LIN {X 0,Y 421.841,Z 771.476,A -85,B 0,C 180,E1 10209.107,E2 10209.107} C_VEL
LIN {X 0,Y 405.011,Z 742.574,A -85,B 0,C 180,E1 10212.582,E2 10212.582} C_VEL
LIN {X 0,Y 403.08,Z 737.44,A -85,B 0,C 180,E1 10213.086,E2 10213.086} C_VEL
LIN {X 0,Y 403.121,Z 737.44,A -85,B 0,C 180,E1 10218.689,E2 10218.689} C_VEL
LIN {X 0,Y 403.149,Z 737.44,A -85,B 0,C 180,E1 10225.725,E2 10225.725} C_VEL
LIN {X 0,Y 403.287,Z 737.44,A -85,B 0,C 180,E1 10230.797,E2 10230.797} C_VEL
LIN {X 0,Y 403.605,Z 737.44,A -85,B 0,C 180,E1 10237.976,E2 10237.976} C_VEL
LIN {X 0,Y 403.898,Z 737.44,A -85,B 0,C 180,E1 10244.795,E2 10244.795} C_VEL
LIN {X 0,Y 404.153,Z 737.44,A -85,B 0,C 180,E1 10251.389,E2 10251.389} C_VEL
LIN {X 0,Y 404.396,Z 737.44,A -85,B 0,C 180,E1 10257.86,E2 10257.86} C_VEL
LIN {X 0,Y 404.246,Z 737.44,A -85,B 0,C 180,E1 10264.301,E2 10264.301} C_VEL
LIN {X 0,Y 403.948,Z 737.44,A -85,B 0,C 180,E1 10270.806,E2 10270.806} C_VEL
LIN {X 0,Y 403.703,Z 737.44,A -85,B 0,C 180,E1 10277.463,E2 10277.463} C_VEL
LIN {X 0,Y 403.474,Z 737.44,A -85,B 0,C 180,E1 10284.383,E2 10284.383} C_VEL
LIN {X 0,Y 403.248,Z 737.44,A -85,B 0,C 180,E1 10291.714,E2 10291.714} C_VEL
LIN {X 0,Y 403.323,Z 738.232,A -85,B 0,C 180,E1 10296.977,E2 10296.977} C_VEL
LIN {X 0,Y 406.403,Z 743.737,A -85,B 0,C 180,E1 10297.606,E2 10297.606} C_VEL
LIN {X 0,Y 427.744,Z 781.818,A -85,B 0,C 180,E1 10301.54,E2 10301.54} C_VEL
LIN {X 0,Y 442.603,Z 815.8,A -85,B 0,C 180,E1 10304.217,E2 10304.217} C_VEL
LIN {X 0,Y 438.64,Z 858.115,A -85,B 0,C 180,E1 10305.69,E2 10305.69} C_VEL
LIN {X 0,Y 433.492,Z 898.592,A -85,B 0,C 180,E1 10307.86,E2 10307.86} C_VEL
LIN {X 0,Y 427.452,Z 938.526,A -85,B 0,C 180,E1 10310.854,E2 10310.854} C_VEL
LIN {X 0,Y 420.959,Z 978.52,A -85,B 0,C 180,E1 10314.869,E2 10314.869} C_VEL
LIN {X 0,Y 415.665,Z 1011.15,A -85,B 0,C 180,E1 10319.101,E2 10319.101} C_VEL
LIN {X 0,Y 411.27,Z 1038.766,A -85,B 0,C 180,E1 10323.784,E2 10323.784} C_VEL
LIN {X 0,Y 408.924,Z 1055.24,A -85,B 0,C 180,E1 10327.316,E2 10327.316} C_VEL
LIN {X 0,Y 403.983,Z 1063.313,A -85,B 0,C 180,E1 10329.395,E2 10329.395} C_VEL
LIN {X 0,Y 399.077,Z 1070.528,A -85,B 0,C 180,E1 10331.574,E2 10331.574} C_VEL
LIN {X 0,Y 397.48,Z 1085.683,A -85,B 0,C 180,E1 10337.349,E2 10337.349} C_VEL
LIN {X 0,Y 396.899,Z 1094.4,A -85,B 0,C 180,E1 10342.658,E2 10342.658} C_VEL
LIN {X 0,Y 396.783,Z 1098.451,A -85,B 0,C 180,E1 10347.813,E2 10347.813} C_VEL
LIN {X 0,Y 396.696,Z 1098.441,A -85,B 0,C 180,E1 10352.187,E2 10352.187} C_VEL
LIN {X 0,Y 396.89,Z 1094.411,A -85,B 0,C 180,E1 10357.332,E2 10357.332} C_VEL
LIN {X 0,Y 397.455,Z 1085.675,A -85,B 0,C 180,E1 10362.652,E2 10362.652} C_VEL
LIN {X 0,Y 398.842,Z 1071.644,A -85,B 0,C 180,E1 10368.064,E2 10368.064} C_VEL
LIN {X 0,Y 401.384,Z 1052.51,A -85,B 0,C 180,E1 10373.331,E2 10373.331} C_VEL
LIN {X 0,Y 405.144,Z 1028.089,A -85,B 0,C 180,E1 10378.34,E2 10378.34} C_VEL
LIN {X 0,Y 410.502,Z 996.087,A -85,B 0,C 180,E1 10383.284,E2 10383.284} C_VEL
LIN {X 0,Y 417.164,Z 957.356,A -85,B 0,C 180,E1 10387.871,E2 10387.871} C_VEL
LIN {X 0,Y 423.856,Z 917.641,A -85,B 0,C 180,E1 10391.397,E2 10391.397} C_VEL
LIN {X 0,Y 430,Z 877.022,A -85,B 0,C 180,E1 10394.013,E2 10394.013} C_VEL
LIN {X 0,Y 435.089,Z 835.418,A -85,B 0,C 180,E1 10395.826,E2 10395.826} C_VEL
LIN {X 0,Y 436.104,Z 818.323,A -85,B 0,C 180,E1 10396.409,E2 10396.409} C_VEL
LIN {X 0,Y 419.344,Z 779.704,A -85,B 0,C 180,E1 10399.601,E2 10399.601} C_VEL
LIN {X 0,Y 400.478,Z 747.677,A -85,B 0,C 180,E1 10403.212,E2 10403.212} C_VEL
LIN {X 0,Y 395.409,Z 739.078,A -85,B 0,C 180,E1 10404.289,E2 10404.289} C_VEL
LIN {X 0,Y 395.252,Z 737.44,A -85,B 0,C 180,E1 10404.437,E2 10404.437} C_VEL
LIN {X 0,Y 395.382,Z 737.44,A -85,B 0,C 180,E1 10411.728,E2 10411.728} C_VEL
LIN {X 0,Y 395.629,Z 737.44,A -85,B 0,C 180,E1 10417.496,E2 10417.496} C_VEL
LIN {X 0,Y 395.787,Z 737.44,A -85,B 0,C 180,E1 10424.464,E2 10424.464} C_VEL
LIN {X 0,Y 396.151,Z 737.44,A -85,B 0,C 180,E1 10431.202,E2 10431.202} C_VEL
LIN {X 0,Y 396.597,Z 737.44,A -85,B 0,C 180,E1 10437.807,E2 10437.807} C_VEL
LIN {X 0,Y 396.428,Z 737.44,A -85,B 0,C 180,E1 10444.375,E2 10444.375} C_VEL
LIN {X 0,Y 396.073,Z 737.44,A -85,B 0,C 180,E1 10451.012,E2 10451.012} C_VEL
LIN {X 0,Y 395.827,Z 737.44,A -85,B 0,C 180,E1 10457.81,E2 10457.81} C_VEL
LIN {X 0,Y 395.507,Z 737.44,A -85,B 0,C 180,E1 10464.894,E2 10464.894} C_VEL
LIN {X 0,Y 395.372,Z 737.44,A -85,B 0,C 180,E1 10469.846,E2 10469.846} C_VEL
LIN {X 0,Y 395.152,Z 737.44,A -85,B 0,C 180,E1 10476.429,E2 10476.429} C_VEL
LIN {X 0,Y 395.184,Z 737.44,A -85,B 0,C 180,E1 10483.586,E2 10483.586} C_VEL
LIN {X 0,Y 395.265,Z 737.646,A -85,B 0,C 180,E1 10485.607,E2 10485.607} C_VEL
LIN {X 0,Y 397.662,Z 743.14,A -85,B 0,C 180,E1 10486.146,E2 10486.146} C_VEL
LIN {X 0,Y 414.525,Z 771.892,A -85,B 0,C 180,E1 10489.793,E2 10489.793} C_VEL
LIN {X 0,Y 428.558,Z 803.812,A -85,B 0,C 180,E1 10493.591,E2 10493.591} C_VEL
LIN {X 0,Y 430.654,Z 811.626,A -85,B 0,C 180,E1 10494.448,E2 10494.448} C_VEL
LIN {X 0,Y 424.989,Z 845.077,A -85,B 0,C 180,E1 10496.949,E2 10496.949} C_VEL
LIN {X 0,Y 418.349,Z 876.019,A -85,B 0,C 180,E1 10500.272,E2 10500.272} C_VEL
LIN {X 0,Y 411.534,Z 902.916,A -85,B 0,C 180,E1 10504.351,E2 10504.351} C_VEL
LIN {X 0,Y 406.088,Z 923.632,A -85,B 0,C 180,E1 10508.73,E2 10508.73} C_VEL
LIN {X 0,Y 401.972,Z 940.182,A -85,B 0,C 180,E1 10513.677,E2 10513.677} C_VEL
LIN {X 0,Y 399.383,Z 952.165,A -85,B 0,C 180,E1 10519.074,E2 10519.074} C_VEL
LIN {X 0,Y 398.349,Z 958.027,A -85,B 0,C 180,E1 10523.453,E2 10523.453} C_VEL
LIN {X 0,Y 398.03,Z 960.855,A -85,B 0,C 180,E1 10527.82,E2 10527.82} C_VEL
LIN {X 0,Y 398.031,Z 960.817,A -85,B 0,C 180,E1 10532.18,E2 10532.18} C_VEL
LIN {X 0,Y 398.524,Z 956.746,A -85,B 0,C 180,E1 10537.641,E2 10537.641} C_VEL
LIN {X 0,Y 400.243,Z 947.761,A -85,B 0,C 180,E1 10543.118,E2 10543.118} C_VEL
LIN {X 0,Y 403.75,Z 933.079,A -85,B 0,C 180,E1 10548.587,E2 10548.587} C_VEL
LIN {X 0,Y 408.801,Z 913.656,A -85,B 0,C 180,E1 10553.461,E2 10553.461} C_VEL
LIN {X 0,Y 414.975,Z 889.704,A -85,B 0,C 180,E1 10557.721,E2 10557.721} C_VEL
LIN {X 0,Y 421.419,Z 862.286,A -85,B 0,C 180,E1 10561.244,E2 10561.244} C_VEL
LIN {X 0,Y 427.498,Z 831.792,A -85,B 0,C 180,E1 10564.053,E2 10564.053} C_VEL
LIN {X 0,Y 430.432,Z 808.17,A -85,B 0,C 180,E1 10565.755,E2 10565.755} C_VEL
LIN {X 0,Y 415.605,Z 774.12,A -85,B 0,C 180,E1 10569.852,E2 10569.852} C_VEL
LIN {X 0,Y 397.852,Z 743.365,A -85,B 0,C 180,E1 10573.708,E2 10573.708} C_VEL
LIN {X 0,Y 395.377,Z 739.015,A -85,B 0,C 180,E1 10574.232,E2 10574.232} C_VEL
LIN {X 0,Y 395.222,Z 737.44,A -85,B 0,C 180,E1 10574.384,E2 10574.384} C_VEL
LIN {X 0,Y 395.2,Z 737.44,A -85,B 0,C 180,E1 10580.013,E2 10580.013} C_VEL
LIN {X 0,Y 395.222,Z 737.44,A -85,B 0,C 180,E1 10587.578,E2 10587.578} C_VEL
LIN {X 0,Y 395.401,Z 737.44,A -85,B 0,C 180,E1 10592.655,E2 10592.655} C_VEL
LIN {X 0,Y 395.782,Z 737.44,A -85,B 0,C 180,E1 10599.87,E2 10599.87} C_VEL
LIN {X 0,Y 396.097,Z 737.44,A -85,B 0,C 180,E1 10606.749,E2 10606.749} C_VEL
LIN {X 0,Y 396.295,Z 737.44,A -85,B 0,C 180,E1 10613.425,E2 10613.425} C_VEL
LIN {X 0,Y 396.616,Z 737.44,A -85,B 0,C 180,E1 10620.006,E2 10620.006} C_VEL
LIN {X 0,Y 396.298,Z 737.44,A -85,B 0,C 180,E1 10626.642,E2 10626.642} C_VEL
LIN {X 0,Y 395.952,Z 737.44,A -85,B 0,C 180,E1 10633.268,E2 10633.268} C_VEL
LIN {X 0,Y 395.718,Z 737.44,A -85,B 0,C 180,E1 10640.146,E2 10640.146} C_VEL
LIN {X 0,Y 395.425,Z 737.44,A -85,B 0,C 180,E1 10647.356,E2 10647.356} C_VEL
LIN {X 0,Y 395.261,Z 737.44,A -85,B 0,C 180,E1 10655.072,E2 10655.072} C_VEL
LIN {X 0,Y 395.239,Z 737.44,A -85,B 0,C 180,E1 10655.647,E2 10655.647} C_VEL
LIN {X 0,Y 397.67,Z 743.102,A -85,B 0,C 180,E1 10656.218,E2 10656.218} C_VEL
LIN {X 0,Y 415.703,Z 773.164,A -85,B 0,C 180,E1 10659.745,E2 10659.745} C_VEL
LIN {X 0,Y 428.985,Z 800.821,A -85,B 0,C 180,E1 10662.195,E2 10662.195} C_VEL
LIN {X 0,Y 436.269,Z 820.576,A -85,B 0,C 180,E1 10663.692,E2 10663.692} C_VEL
LIN {X 0,Y 431.56,Z 864.796,A -85,B 0,C 180,E1 10665.359,E2 10665.359} C_VEL
LIN {X 0,Y 425.309,Z 908.643,A -85,B 0,C 180,E1 10667.939,E2 10667.939} C_VEL
LIN {X 0,Y 418.55,Z 949.549,A -85,B 0,C 180,E1 10671.352,E2 10671.352} C_VEL
LIN {X 0,Y 411.952,Z 987.61,A -85,B 0,C 180,E1 10675.612,E2 10675.612} C_VEL
LIN {X 0,Y 406.631,Z 1019.135,A -85,B 0,C 180,E1 10680.133,E2 10680.133} C_VEL
LIN {X 0,Y 402.24,Z 1046.295,A -85,B 0,C 180,E1 10685.252,E2 10685.252} C_VEL
LIN {X 0,Y 399.278,Z 1068.312,A -85,B 0,C 180,E1 10690.867,E2 10690.867} C_VEL
LIN {X 0,Y 399.077,Z 1070.528,A -85,B 0,C 180,E1 10691.574,E2 10691.574} C_VEL
LIN {X 0,Y 395.94,Z 1075.45,A -85,B 0,C 180,E1 10693.276,E2 10693.276} C_VEL
LIN {X 0,Y 390.017,Z 1081.554,A -85,B 0,C 180,E1 10695.892,E2 10695.892} C_VEL
LIN {X 0,Y 389.867,Z 1082.242,A -85,B 0,C 180,E1 10696.198,E2 10696.198} C_VEL
LIN {X 0,Y 389.186,Z 1091.15,A -85,B 0,C 180,E1 10701.048,E2 10701.048} C_VEL
LIN {X 0,Y 388.942,Z 1095.94,A -85,B 0,C 180,E1 10705.535,E2 10705.535} C_VEL
LIN {X 0,Y 388.979,Z 1097.538,A -85,B 0,C 180,E1 10710,E2 10710} C_VEL
LIN {X 0,Y 388.927,Z 1095.938,A -85,B 0,C 180,E1 10714.465,E2 10714.465} C_VEL
LIN {X 0,Y 389.299,Z 1089.365,A -85,B 0,C 180,E1 10720.079,E2 10720.079} C_VEL
LIN {X 0,Y 390.296,Z 1077.552,A -85,B 0,C 180,E1 10725.755,E2 10725.755} C_VEL
LIN {X 0,Y 392.312,Z 1060.229,A -85,B 0,C 180,E1 10731.353,E2 10731.353} C_VEL
LIN {X 0,Y 396.104,Z 1035.93,A -85,B 0,C 180,E1 10736.994,E2 10736.994} C_VEL
LIN {X 0,Y 401.278,Z 1005.115,A -85,B 0,C 180,E1 10742.313,E2 10742.313} C_VEL
LIN {X 0,Y 407.929,Z 969.196,A -85,B 0,C 180,E1 10747.066,E2 10747.066} C_VEL
LIN {X 0,Y 414.997,Z 930.635,A -85,B 0,C 180,E1 10750.917,E2 10750.917} C_VEL
LIN {X 0,Y 421.67,Z 890.291,A -85,B 0,C 180,E1 10753.88,E2 10753.88} C_VEL
LIN {X 0,Y 427.438,Z 848.09,A -85,B 0,C 180,E1 10756.03,E2 10756.03} C_VEL
LIN {X 0,Y 429.943,Z 821.334,A -85,B 0,C 180,E1 10757.002,E2 10757.002} C_VEL
LIN {X 0,Y 414.605,Z 784.809,A -85,B 0,C 180,E1 10760.106,E2 10760.106} C_VEL
LIN {X 0,Y 394.236,Z 749.739,A -85,B 0,C 180,E1 10764.167,E2 10764.167} C_VEL
LIN {X 0,Y 387.474,Z 739.028,A -85,B 0,C 180,E1 10765.661,E2 10765.661} C_VEL
LIN {X 0,Y 387.292,Z 737.44,A -85,B 0,C 180,E1 10765.839,E2 10765.839} C_VEL
LIN {X 0,Y 387.509,Z 737.44,A -85,B 0,C 180,E1 10772.037,E2 10772.037} C_VEL
LIN {X 0,Y 387.819,Z 737.44,A -85,B 0,C 180,E1 10779.541,E2 10779.541} C_VEL
LIN {X 0,Y 387.94,Z 737.44,A -85,B 0,C 180,E1 10786.453,E2 10786.453} C_VEL
LIN {X 0,Y 388.406,Z 737.44,A -85,B 0,C 180,E1 10793.279,E2 10793.279} C_VEL
LIN {X 0,Y 388.708,Z 737.44,A -85,B 0,C 180,E1 10799.994,E2 10799.994} C_VEL
LIN {X 0,Y 388.394,Z 737.44,A -85,B 0,C 180,E1 10806.709,E2 10806.709} C_VEL
LIN {X 0,Y 388.017,Z 737.44,A -85,B 0,C 180,E1 10813.532,E2 10813.532} C_VEL
LIN {X 0,Y 387.776,Z 737.44,A -85,B 0,C 180,E1 10820.564,E2 10820.564} C_VEL
LIN {X 0,Y 387.493,Z 737.44,A -85,B 0,C 180,E1 10827.951,E2 10827.951} C_VEL
LIN {X 0,Y 387.292,Z 737.44,A -85,B 0,C 180,E1 10834.823,E2 10834.823} C_VEL
LIN {X 0,Y 387.166,Z 737.44,A -85,B 0,C 180,E1 10842.014,E2 10842.014} C_VEL
LIN {X 0,Y 387.319,Z 737.534,A -85,B 0,C 180,E1 10844.215,E2 10844.215} C_VEL
LIN {X 0,Y 389.582,Z 742.952,A -85,B 0,C 180,E1 10844.756,E2 10844.756} C_VEL
LIN {X 0,Y 404.932,Z 768.164,A -85,B 0,C 180,E1 10848.198,E2 10848.198} C_VEL
LIN {X 0,Y 418.919,Z 798.421,A -85,B 0,C 180,E1 10851.948,E2 10851.948} C_VEL
LIN {X 0,Y 424.538,Z 812.7,A -85,B 0,C 180,E1 10853.767,E2 10853.767} C_VEL
LIN {X 0,Y 418.814,Z 845.679,A -85,B 0,C 180,E1 10856.264,E2 10856.264} C_VEL
LIN {X 0,Y 412.303,Z 875.144,A -85,B 0,C 180,E1 10859.428,E2 10859.428} C_VEL
LIN {X 0,Y 405.399,Z 901.689,A -85,B 0,C 180,E1 10863.375,E2 10863.375} C_VEL
LIN {X 0,Y 399.204,Z 923.93,A -85,B 0,C 180,E1 10868.029,E2 10868.029} C_VEL
LIN {X 0,Y 394.663,Z 940.979,A -85,B 0,C 180,E1 10873.132,E2 10873.132} C_VEL
LIN {X 0,Y 391.738,Z 953.55,A -85,B 0,C 180,E1 10878.858,E2 10878.858} C_VEL
LIN {X 0,Y 390.595,Z 959.39,A -85,B 0,C 180,E1 10883.323,E2 10883.323} C_VEL
LIN {X 0,Y 390.259,Z 962.203,A -85,B 0,C 180,E1 10887.777,E2 10887.777} C_VEL
LIN {X 0,Y 390.26,Z 962.166,A -85,B 0,C 180,E1 10892.223,E2 10892.223} C_VEL
LIN {X 0,Y 390.819,Z 958.112,A -85,B 0,C 180,E1 10897.793,E2 10897.793} C_VEL
LIN {X 0,Y 392.637,Z 949.163,A -85,B 0,C 180,E1 10903.377,E2 10903.377} C_VEL
LIN {X 0,Y 396.354,Z 934.52,A -85,B 0,C 180,E1 10908.946,E2 10908.946} C_VEL
LIN {X 0,Y 401.689,Z 915.169,A -85,B 0,C 180,E1 10913.902,E2 10913.902} C_VEL
LIN {X 0,Y 408.132,Z 891.302,A -85,B 0,C 180,E1 10918.227,E2 10918.227} C_VEL
LIN {X 0,Y 414.873,Z 864.009,A -85,B 0,C 180,E1 10921.794,E2 10921.794} C_VEL
LIN {X 0,Y 421.198,Z 833.59,A -85,B 0,C 180,E1 10924.65,E2 10924.65} C_VEL
LIN {X 0,Y 424.271,Z 811.845,A -85,B 0,C 180,E1 10926.237,E2 10926.237} C_VEL
LIN {X 0,Y 410.562,Z 779.323,A -85,B 0,C 180,E1 10930.296,E2 10930.296} C_VEL
LIN {X 0,Y 394,Z 749.53,A -85,B 0,C 180,E1 10934.172,E2 10934.172} C_VEL
LIN {X 0,Y 387.441,Z 739.105,A -85,B 0,C 180,E1 10935.612,E2 10935.612} C_VEL
LIN {X 0,Y 387.291,Z 737.44,A -85,B 0,C 180,E1 10935.832,E2 10935.832} C_VEL
LIN {X 0,Y 387.222,Z 737.44,A -85,B 0,C 180,E1 10941.442,E2 10941.442} C_VEL
LIN {X 0,Y 387.265,Z 737.44,A -85,B 0,C 180,E1 10946.827,E2 10946.827} C_VEL
LIN {X 0,Y 387.493,Z 737.44,A -85,B 0,C 180,E1 10953.98,E2 10953.98} C_VEL
LIN {X 0,Y 387.839,Z 737.44,A -85,B 0,C 180,E1 10959.534,E2 10959.534} C_VEL
LIN {X 0,Y 388.145,Z 737.44,A -85,B 0,C 180,E1 10966.472,E2 10966.472} C_VEL
LIN {X 0,Y 388.403,Z 737.44,A -85,B 0,C 180,E1 10973.291,E2 10973.291} C_VEL
LIN {X 0,Y 388.721,Z 737.44,A -85,B 0,C 180,E1 10980.006,E2 10980.006} C_VEL
LIN {X 0,Y 388.409,Z 737.44,A -85,B 0,C 180,E1 10986.721,E2 10986.721} C_VEL
LIN {X 0,Y 388.023,Z 737.44,A -85,B 0,C 180,E1 10993.544,E2 10993.544} C_VEL
LIN {X 0,Y 387.746,Z 737.44,A -85,B 0,C 180,E1 11000.578,E2 11000.578} C_VEL
LIN {X 0,Y 387.511,Z 737.44,A -85,B 0,C 180,E1 11007.963,E2 11007.963} C_VEL
LIN {X 0,Y 387.33,Z 738.182,A -85,B 0,C 180,E1 11014.305,E2 11014.305} C_VEL
LIN {X 0,Y 390.362,Z 743.645,A -85,B 0,C 180,E1 11015.008,E2 11015.008} C_VEL
LIN {X 0,Y 410.275,Z 776.907,A -85,B 0,C 180,E1 11019.087,E2 11019.087} C_VEL
LIN {X 0,Y 423.666,Z 805.087,A -85,B 0,C 180,E1 11021.665,E2 11021.665} C_VEL
LIN {X 0,Y 430.005,Z 823.304,A -85,B 0,C 180,E1 11023.092,E2 11023.092} C_VEL
LIN {X 0,Y 425.026,Z 866.64,A -85,B 0,C 180,E1 11024.801,E2 11024.801} C_VEL
LIN {X 0,Y 418.758,Z 908.301,A -85,B 0,C 180,E1 11027.317,E2 11027.317} C_VEL
LIN {X 0,Y 411.734,Z 948.535,A -85,B 0,C 180,E1 11030.731,E2 11030.731} C_VEL
LIN {X 0,Y 404.856,Z 985.634,A -85,B 0,C 180,E1 11034.955,E2 11034.955} C_VEL
LIN {X 0,Y 398.978,Z 1018.404,A -85,B 0,C 180,E1 11039.815,E2 11039.815} C_VEL
LIN {X 0,Y 394.494,Z 1045.535,A -85,B 0,C 180,E1 11045.029,E2 11045.029} C_VEL
LIN {X 0,Y 391.418,Z 1067.482,A -85,B 0,C 180,E1 11050.759,E2 11050.759} C_VEL
LIN {X 0,Y 389.867,Z 1082.242,A -85,B 0,C 180,E1 11056.198,E2 11056.198} C_VEL
LIN {X 0,Y 387.079,Z 1085.8,A -85,B 0,C 180,E1 11058.014,E2 11058.014} C_VEL
LIN {X 0,Y 381.354,Z 1090.058,A -85,B 0,C 180,E1 11061.13,E2 11061.13} C_VEL
LIN {X 0,Y 381.154,Z 1094.572,A -85,B 0,C 180,E1 11065.443,E2 11065.443} C_VEL
LIN {X 0,Y 381.219,Z 1096.194,A -85,B 0,C 180,E1 11070,E2 11070} C_VEL
LIN {X 0,Y 381.135,Z 1093.584,A -85,B 0,C 180,E1 11075.699,E2 11075.699} C_VEL
LIN {X 0,Y 381.614,Z 1086.021,A -85,B 0,C 180,E1 11081.441,E2 11081.441} C_VEL
LIN {X 0,Y 382.882,Z 1072.845,A -85,B 0,C 180,E1 11087.251,E2 11087.251} C_VEL
LIN {X 0,Y 385.145,Z 1055.038,A -85,B 0,C 180,E1 11092.676,E2 11092.676} C_VEL
LIN {X 0,Y 388.777,Z 1032.212,A -85,B 0,C 180,E1 11097.86,E2 11097.86} C_VEL
LIN {X 0,Y 394.4,Z 1001.797,A -85,B 0,C 180,E1 11103.162,E2 11103.162} C_VEL
LIN {X 0,Y 401.274,Z 966.87,A -85,B 0,C 180,E1 11107.825,E2 11107.825} C_VEL
LIN {X 0,Y 408.421,Z 929.423,A -85,B 0,C 180,E1 11111.613,E2 11111.613} C_VEL
LIN {X 0,Y 415.284,Z 890.253,A -85,B 0,C 180,E1 11114.531,E2 11114.531} C_VEL
LIN {X 0,Y 421.394,Z 847.653,A -85,B 0,C 180,E1 11116.733,E2 11116.733} C_VEL
LIN {X 0,Y 423.515,Z 823.807,A -85,B 0,C 180,E1 11117.649,E2 11117.649} C_VEL
LIN {X 0,Y 410.325,Z 790.912,A -85,B 0,C 180,E1 11120.533,E2 11120.533} C_VEL
LIN {X 0,Y 390.362,Z 755.855,A -85,B 0,C 180,E1 11124.636,E2 11124.636} C_VEL
LIN {X 0,Y 379.526,Z 738.977,A -85,B 0,C 180,E1 11127.137,E2 11127.137} C_VEL
LIN {X 0,Y 379.369,Z 737.44,A -85,B 0,C 180,E1 11127.231,E2 11127.231} C_VEL
LIN {X 0,Y 379.633,Z 737.44,A -85,B 0,C 180,E1 11133.976,E2 11133.976} C_VEL
LIN {X 0,Y 379.903,Z 737.44,A -85,B 0,C 180,E1 11141.404,E2 11141.404} C_VEL
LIN {X 0,Y 380.092,Z 737.44,A -85,B 0,C 180,E1 11148.507,E2 11148.507} C_VEL
LIN {X 0,Y 380.523,Z 737.44,A -85,B 0,C 180,E1 11155.43,E2 11155.43} C_VEL
LIN {X 0,Y 380.806,Z 737.44,A -85,B 0,C 180,E1 11159.994,E2 11159.994} C_VEL
LIN {X 0,Y 380.489,Z 737.44,A -85,B 0,C 180,E1 11166.849,E2 11166.849} C_VEL
LIN {X 0,Y 380.074,Z 737.44,A -85,B 0,C 180,E1 11173.821,E2 11173.821} C_VEL
LIN {X 0,Y 379.798,Z 737.44,A -85,B 0,C 180,E1 11181.016,E2 11181.016} C_VEL
LIN {X 0,Y 379.51,Z 737.44,A -85,B 0,C 180,E1 11188.64,E2 11188.64} C_VEL
LIN {X 0,Y 379.373,Z 737.44,A -85,B 0,C 180,E1 11193.956,E2 11193.956} C_VEL
LIN {X 0,Y 379.301,Z 737.44,A -85,B 0,C 180,E1 11202.172,E2 11202.172} C_VEL
LIN {X 0,Y 379.325,Z 737.611,A -85,B 0,C 180,E1 11202.715,E2 11202.715} C_VEL
LIN {X 0,Y 381.745,Z 743.09,A -85,B 0,C 180,E1 11203.325,E2 11203.325} C_VEL
LIN {X 0,Y 397.003,Z 767.444,A -85,B 0,C 180,E1 11206.902,E2 11206.902} C_VEL
LIN {X 0,Y 410.809,Z 796.567,A -85,B 0,C 180,E1 11210.694,E2 11210.694} C_VEL
LIN {X 0,Y 418.16,Z 817.191,A -85,B 0,C 180,E1 11213.308,E2 11213.308} C_VEL
LIN {X 0,Y 411.742,Z 850.959,A -85,B 0,C 180,E1 11215.993,E2 11215.993} C_VEL
LIN {X 0,Y 404.723,Z 880.357,A -85,B 0,C 180,E1 11219.341,E2 11219.341} C_VEL
LIN {X 0,Y 397.578,Z 906.104,A -85,B 0,C 180,E1 11223.413,E2 11223.413} C_VEL
LIN {X 0,Y 391.31,Z 927.634,A -85,B 0,C 180,E1 11228.185,E2 11228.185} C_VEL
LIN {X 0,Y 386.764,Z 943.995,A -85,B 0,C 180,E1 11233.39,E2 11233.39} C_VEL
LIN {X 0,Y 384.071,Z 954.935,A -85,B 0,C 180,E1 11238.633,E2 11238.633} C_VEL
LIN {X 0,Y 382.85,Z 960.75,A -85,B 0,C 180,E1 11243.187,E2 11243.187} C_VEL
LIN {X 0,Y 382.496,Z 963.55,A -85,B 0,C 180,E1 11247.732,E2 11247.732} C_VEL
LIN {X 0,Y 382.497,Z 963.513,A -85,B 0,C 180,E1 11252.269,E2 11252.269} C_VEL
LIN {X 0,Y 383.102,Z 959.478,A -85,B 0,C 180,E1 11257.951,E2 11257.951} C_VEL
LIN {X 0,Y 385.049,Z 950.557,A -85,B 0,C 180,E1 11263.646,E2 11263.646} C_VEL
LIN {X 0,Y 388.978,Z 935.949,A -85,B 0,C 180,E1 11269.32,E2 11269.32} C_VEL
LIN {X 0,Y 394.929,Z 915.353,A -85,B 0,C 180,E1 11274.639,E2 11274.639} C_VEL
LIN {X 0,Y 401.79,Z 891.115,A -85,B 0,C 180,E1 11279.022,E2 11279.022} C_VEL
LIN {X 0,Y 408.851,Z 863.362,A -85,B 0,C 180,E1 11282.633,E2 11282.633} C_VEL
LIN {X 0,Y 415.826,Z 830.778,A -85,B 0,C 180,E1 11285.63,E2 11285.63} C_VEL
LIN {X 0,Y 418.035,Z 815.331,A -85,B 0,C 180,E1 11286.762,E2 11286.762} C_VEL
LIN {X 0,Y 405.1,Z 783.565,A -85,B 0,C 180,E1 11290.866,E2 11290.866} C_VEL
LIN {X 0,Y 389.644,Z 755.049,A -85,B 0,C 180,E1 11294.75,E2 11294.75} C_VEL
LIN {X 0,Y 381.124,Z 742.334,A -85,B 0,C 180,E1 11296.698,E2 11296.698} C_VEL
LIN {X 0,Y 379.374,Z 737.44,A -85,B 0,C 180,E1 11297.291,E2 11297.291} C_VEL
LIN {X 0,Y 379.236,Z 737.44,A -85,B 0,C 180,E1 11303.225,E2 11303.225} C_VEL
LIN {X 0,Y 379.37,Z 737.44,A -85,B 0,C 180,E1 11308.758,E2 11308.758} C_VEL
LIN {X 0,Y 379.687,Z 737.44,A -85,B 0,C 180,E1 11316.509,E2 11316.509} C_VEL
LIN {X 0,Y 380.077,Z 737.44,A -85,B 0,C 180,E1 11323.817,E2 11323.817} C_VEL
LIN {X 0,Y 380.348,Z 737.44,A -85,B 0,C 180,E1 11331.267,E2 11331.267} C_VEL
LIN {X 0,Y 380.699,Z 737.44,A -85,B 0,C 180,E1 11337.727,E2 11337.727} C_VEL
LIN {X 0,Y 380.791,Z 737.44,A -85,B 0,C 180,E1 11342.284,E2 11342.284} C_VEL
LIN {X 0,Y 380.312,Z 737.44,A -85,B 0,C 180,E1 11349.168,E2 11349.168} C_VEL
LIN {X 0,Y 379.961,Z 737.44,A -85,B 0,C 180,E1 11356.201,E2 11356.201} C_VEL
LIN {X 0,Y 379.681,Z 737.44,A -85,B 0,C 180,E1 11363.505,E2 11363.505} C_VEL
LIN {X 0,Y 379.509,Z 737.44,A -85,B 0,C 180,E1 11368.639,E2 11368.639} C_VEL
LIN {X 0,Y 379.402,Z 737.821,A -85,B 0,C 180,E1 11372.82,E2 11372.82} C_VEL
LIN {X 0,Y 382.098,Z 743.376,A -85,B 0,C 180,E1 11373.512,E2 11373.512} C_VEL
LIN {X 0,Y 400.478,Z 772.857,A -85,B 0,C 180,E1 11377.523,E2 11377.523} C_VEL
LIN {X 0,Y 415.683,Z 802.707,A -85,B 0,C 180,E1 11380.568,E2 11380.568} C_VEL
LIN {X 0,Y 423.816,Z 825.935,A -85,B 0,C 180,E1 11382.487,E2 11382.487} C_VEL
LIN {X 0,Y 418.64,Z 867.719,A -85,B 0,C 180,E1 11384.19,E2 11384.19} C_VEL
LIN {X 0,Y 412.01,Z 909.261,A -85,B 0,C 180,E1 11386.768,E2 11386.768} C_VEL
LIN {X 0,Y 404.786,Z 948.275,A -85,B 0,C 180,E1 11390.155,E2 11390.155} C_VEL
LIN {X 0,Y 397.715,Z 984.35,A -85,B 0,C 180,E1 11394.345,E2 11394.345} C_VEL
LIN {X 0,Y 391.522,Z 1016.979,A -85,B 0,C 180,E1 11399.318,E2 11399.318} C_VEL
LIN {X 0,Y 386.716,Z 1044.741,A -85,B 0,C 180,E1 11404.801,E2 11404.801} C_VEL
LIN {X 0,Y 383.628,Z 1065.875,A -85,B 0,C 180,E1 11410.393,E2 11410.393} C_VEL
LIN {X 0,Y 382.014,Z 1081.452,A -85,B 0,C 180,E1 11416.244,E2 11416.244} C_VEL
LIN {X 0,Y 381.354,Z 1090.058,A -85,B 0,C 180,E1 11421.13,E2 11421.13} C_VEL
LIN {X 0,Y 378.722,Z 1092.035,A -85,B 0,C 180,E1 11423.051,E2 11423.051} C_VEL
LIN {X 0,Y 373.307,Z 1093.708,A -85,B 0,C 180,E1 11426.307,E2 11426.307} C_VEL
LIN {X 0,Y 373.432,Z 1094.845,A -85,B 0,C 180,E1 11430,E2 11430} C_VEL
LIN {X 0,Y 373.35,Z 1092.422,A -85,B 0,C 180,E1 11435.559,E2 11435.559} C_VEL
LIN {X 0,Y 373.675,Z 1086.456,A -85,B 0,C 180,E1 11440.505,E2 11440.505} C_VEL
LIN {X 0,Y 374.775,Z 1074.317,A -85,B 0,C 180,E1 11446.426,E2 11446.426} C_VEL
LIN {X 0,Y 377.037,Z 1056.535,A -85,B 0,C 180,E1 11452.258,E2 11452.258} C_VEL
LIN {X 0,Y 381.068,Z 1031.75,A -85,B 0,C 180,E1 11458.151,E2 11458.151} C_VEL
LIN {X 0,Y 387.191,Z 1000.551,A -85,B 0,C 180,E1 11463.749,E2 11463.749} C_VEL
LIN {X 0,Y 394.236,Z 966.503,A -85,B 0,C 180,E1 11468.398,E2 11468.398} C_VEL
LIN {X 0,Y 401.948,Z 928.333,A -85,B 0,C 180,E1 11472.321,E2 11472.321} C_VEL
LIN {X 0,Y 409.226,Z 888.74,A -85,B 0,C 180,E1 11475.292,E2 11475.292} C_VEL
LIN {X 0,Y 415.42,Z 847.386,A -85,B 0,C 180,E1 11477.451,E2 11477.451} C_VEL
LIN {X 0,Y 417.462,Z 826.806,A -85,B 0,C 180,E1 11478.252,E2 11478.252} C_VEL
LIN {X 0,Y 405.084,Z 794.944,A -85,B 0,C 180,E1 11481.153,E2 11481.153} C_VEL
LIN {X 0,Y 386.294,Z 761.703,A -85,B 0,C 180,E1 11485.164,E2 11485.164} C_VEL
LIN {X 0,Y 373.537,Z 742.762,A -85,B 0,C 180,E1 11488.199,E2 11488.199} C_VEL
LIN {X 0,Y 371.495,Z 737.44,A -85,B 0,C 180,E1 11488.852,E2 11488.852} C_VEL
LIN {X 0,Y 371.737,Z 737.44,A -85,B 0,C 180,E1 11495.962,E2 11495.962} C_VEL
LIN {X 0,Y 371.942,Z 737.44,A -85,B 0,C 180,E1 11500.991,E2 11500.991} C_VEL
LIN {X 0,Y 372.151,Z 737.44,A -85,B 0,C 180,E1 11508.258,E2 11508.258} C_VEL
LIN {X 0,Y 372.611,Z 737.44,A -85,B 0,C 180,E1 11515.333,E2 11515.333} C_VEL
LIN {X 0,Y 372.904,Z 737.44,A -85,B 0,C 180,E1 11519.994,E2 11519.994} C_VEL
LIN {X 0,Y 372.558,Z 737.44,A -85,B 0,C 180,E1 11526.996,E2 11526.996} C_VEL
LIN {X 0,Y 372.131,Z 737.44,A -85,B 0,C 180,E1 11534.122,E2 11534.122} C_VEL
LIN {X 0,Y 371.824,Z 737.44,A -85,B 0,C 180,E1 11541.489,E2 11541.489} C_VEL
LIN {X 0,Y 371.61,Z 737.44,A -85,B 0,C 180,E1 11546.616,E2 11546.616} C_VEL
LIN {X 0,Y 371.464,Z 737.44,A -85,B 0,C 180,E1 11551.985,E2 11551.985} C_VEL
LIN {X 0,Y 371.261,Z 737.44,A -85,B 0,C 180,E1 11559.212,E2 11559.212} C_VEL
LIN {X 0,Y 371.324,Z 737.44,A -85,B 0,C 180,E1 11561.083,E2 11561.083} C_VEL
LIN {X 0,Y 373.607,Z 742.939,A -85,B 0,C 180,E1 11561.718,E2 11561.718} C_VEL
LIN {X 0,Y 376.327,Z 746.655,A -85,B 0,C 180,E1 11562.382,E2 11562.382} C_VEL
LIN {X 0,Y 392.031,Z 772.093,A -85,B 0,C 180,E1 11566.307,E2 11566.307} C_VEL
LIN {X 0,Y 405.201,Z 800.859,A -85,B 0,C 180,E1 11570.188,E2 11570.188} C_VEL
LIN {X 0,Y 411.896,Z 820.393,A -85,B 0,C 180,E1 11572.748,E2 11572.748} C_VEL
LIN {X 0,Y 405.165,Z 853.666,A -85,B 0,C 180,E1 11575.482,E2 11575.482} C_VEL
LIN {X 0,Y 397.721,Z 883.297,A -85,B 0,C 180,E1 11578.961,E2 11578.961} C_VEL
LIN {X 0,Y 390.282,Z 908.812,A -85,B 0,C 180,E1 11583.132,E2 11583.132} C_VEL
LIN {X 0,Y 383.639,Z 930.547,A -85,B 0,C 180,E1 11588.139,E2 11588.139} C_VEL
LIN {X 0,Y 378.795,Z 947.099,A -85,B 0,C 180,E1 11593.753,E2 11593.753} C_VEL
LIN {X 0,Y 376.026,Z 958.03,A -85,B 0,C 180,E1 11599.562,E2 11599.562} C_VEL
LIN {X 0,Y 374.795,Z 963.859,A -85,B 0,C 180,E1 11605.366,E2 11605.366} C_VEL
LIN {X 0,Y 374.795,Z 965.243,A -85,B 0,C 180,E1 11610,E2 11610} C_VEL
LIN {X 0,Y 374.809,Z 963.797,A -85,B 0,C 180,E1 11614.634,E2 11614.634} C_VEL
LIN {X 0,Y 376.035,Z 957.897,A -85,B 0,C 180,E1 11620.439,E2 11620.439} C_VEL
LIN {X 0,Y 379.13,Z 945.997,A -85,B 0,C 180,E1 11626.621,E2 11626.621} C_VEL
LIN {X 0,Y 384.237,Z 928.521,A -85,B 0,C 180,E1 11632.298,E2 11632.298} C_VEL
LIN {X 0,Y 390.562,Z 907.864,A -85,B 0,C 180,E1 11636.949,E2 11636.949} C_VEL
LIN {X 0,Y 397.895,Z 882.335,A -85,B 0,C 180,E1 11641.083,E2 11641.083} C_VEL
LIN {X 0,Y 405.629,Z 851.728,A -85,B 0,C 180,E1 11644.609,E2 11644.609} C_VEL
LIN {X 0,Y 411.869,Z 819.883,A -85,B 0,C 180,E1 11647.202,E2 11647.202} C_VEL
LIN {X 0,Y 400.272,Z 789.162,A -85,B 0,C 180,E1 11651.272,E2 11651.272} C_VEL
LIN {X 0,Y 385.461,Z 760.871,A -85,B 0,C 180,E1 11655.255,E2 11655.255} C_VEL
LIN {X 0,Y 374.171,Z 743.478,A -85,B 0,C 180,E1 11658.034,E2 11658.034} C_VEL
LIN {X 0,Y 371.432,Z 738.639,A -85,B 0,C 180,E1 11658.739,E2 11658.739} C_VEL
LIN {X 0,Y 371.346,Z 737.44,A -85,B 0,C 180,E1 11659.043,E2 11659.043} C_VEL
LIN {X 0,Y 371.302,Z 737.44,A -85,B 0,C 180,E1 11665.201,E2 11665.201} C_VEL
LIN {X 0,Y 371.515,Z 737.44,A -85,B 0,C 180,E1 11670.733,E2 11670.733} C_VEL
LIN {X 0,Y 371.709,Z 737.44,A -85,B 0,C 180,E1 11675.973,E2 11675.973} C_VEL
LIN {X 0,Y 372.009,Z 737.44,A -85,B 0,C 180,E1 11681.007,E2 11681.007} C_VEL
LIN {X 0,Y 372.346,Z 737.44,A -85,B 0,C 180,E1 11688.277,E2 11688.277} C_VEL
LIN {X 0,Y 372.711,Z 737.44,A -85,B 0,C 180,E1 11695.347,E2 11695.347} C_VEL
LIN {X 0,Y 372.875,Z 737.44,A -85,B 0,C 180,E1 11702.333,E2 11702.333} C_VEL
LIN {X 0,Y 372.373,Z 737.44,A -85,B 0,C 180,E1 11709.365,E2 11709.365} C_VEL
LIN {X 0,Y 372.049,Z 737.44,A -85,B 0,C 180,E1 11716.555,E2 11716.555} C_VEL
LIN {X 0,Y 371.709,Z 737.44,A -85,B 0,C 180,E1 11724.04,E2 11724.04} C_VEL
LIN {X 0,Y 371.558,Z 738.242,A -85,B 0,C 180,E1 11731.261,E2 11731.261} C_VEL
LIN {X 0,Y 374.291,Z 743.506,A -85,B 0,C 180,E1 11732.003,E2 11732.003} C_VEL
LIN {X 0,Y 392.937,Z 772.745,A -85,B 0,C 180,E1 11736.318,E2 11736.318} C_VEL
LIN {X 0,Y 409.526,Z 804.65,A -85,B 0,C 180,E1 11739.797,E2 11739.797} C_VEL
LIN {X 0,Y 417.619,Z 828.491,A -85,B 0,C 180,E1 11741.851,E2 11741.851} C_VEL
LIN {X 0,Y 412.247,Z 869.066,A -85,B 0,C 180,E1 11743.57,E2 11743.57} C_VEL
LIN {X 0,Y 405.344,Z 910.062,A -85,B 0,C 180,E1 11746.185,E2 11746.185} C_VEL
LIN {X 0,Y 398.091,Z 947.632,A -85,B 0,C 180,E1 11749.522,E2 11749.522} C_VEL
LIN {X 0,Y 390.621,Z 983.508,A -85,B 0,C 180,E1 11753.767,E2 11753.767} C_VEL
LIN {X 0,Y 384.204,Z 1015.263,A -85,B 0,C 180,E1 11758.702,E2 11758.702} C_VEL
LIN {X 0,Y 379.16,Z 1042.707,A -85,B 0,C 180,E1 11764.263,E2 11764.263} C_VEL
LIN {X 0,Y 375.908,Z 1064.126,A -85,B 0,C 180,E1 11769.98,E2 11769.98} C_VEL
LIN {X 0,Y 374.234,Z 1079.906,A -85,B 0,C 180,E1 11775.952,E2 11775.952} C_VEL
LIN {X 0,Y 373.52,Z 1089.77,A -85,B 0,C 180,E1 11781.844,E2 11781.844} C_VEL
LIN {X 0,Y 373.307,Z 1093.708,A -85,B 0,C 180,E1 11786.307,E2 11786.307} C_VEL
LIN {X 0,Y 370.822,Z 1094.138,A -85,B 0,C 180,E1 11788.288,E2 11788.288} C_VEL
LIN {X 0,Y 365.502,Z 1093.2,A -85,B 0,C 180,E1 11791.626,E2 11791.626} C_VEL
LIN {X 0,Y 365.664,Z 1089.758,A -85,B 0,C 180,E1 11797.135,E2 11797.135} C_VEL
LIN {X 0,Y 366.181,Z 1081.247,A -85,B 0,C 180,E1 11802.888,E2 11802.888} C_VEL
LIN {X 0,Y 367.586,Z 1067.613,A -85,B 0,C 180,E1 11808.677,E2 11808.677} C_VEL
LIN {X 0,Y 370.566,Z 1047.455,A -85,B 0,C 180,E1 11814.691,E2 11814.691} C_VEL
LIN {X 0,Y 375.677,Z 1019.986,A -85,B 0,C 180,E1 11820.76,E2 11820.76} C_VEL
LIN {X 0,Y 382.538,Z 987.364,A -85,B 0,C 180,E1 11826.18,E2 11826.18} C_VEL
LIN {X 0,Y 390.28,Z 951.593,A -85,B 0,C 180,E1 11830.668,E2 11830.668} C_VEL
LIN {X 0,Y 398.405,Z 912.615,A -85,B 0,C 180,E1 11834.287,E2 11834.287} C_VEL
LIN {X 0,Y 405.741,Z 872.043,A -85,B 0,C 180,E1 11836.981,E2 11836.981} C_VEL
LIN {X 0,Y 411.251,Z 829.121,A -85,B 0,C 180,E1 11838.932,E2 11838.932} C_VEL
LIN {X 0,Y 400.202,Z 799.749,A -85,B 0,C 180,E1 11841.719,E2 11841.719} C_VEL
LIN {X 0,Y 381.943,Z 767.126,A -85,B 0,C 180,E1 11845.775,E2 11845.775} C_VEL
LIN {X 0,Y 366.2,Z 743.329,A -85,B 0,C 180,E1 11849.73,E2 11849.73} C_VEL
LIN {X 0,Y 363.657,Z 738.335,A -85,B 0,C 180,E1 11850.484,E2 11850.484} C_VEL
LIN {X 0,Y 363.624,Z 737.44,A -85,B 0,C 180,E1 11850.969,E2 11850.969} C_VEL
LIN {X 0,Y 363.871,Z 737.44,A -85,B 0,C 180,E1 11858.004,E2 11858.004} C_VEL
LIN {X 0,Y 364.124,Z 737.44,A -85,B 0,C 180,E1 11865.548,E2 11865.548} C_VEL
LIN {X 0,Y 364.652,Z 737.44,A -85,B 0,C 180,E1 11872.839,E2 11872.839} C_VEL
LIN {X 0,Y 365.002,Z 737.44,A -85,B 0,C 180,E1 11879.994,E2 11879.994} C_VEL
LIN {X 0,Y 364.649,Z 737.44,A -85,B 0,C 180,E1 11887.148,E2 11887.148} C_VEL
LIN {X 0,Y 364.187,Z 737.44,A -85,B 0,C 180,E1 11894.436,E2 11894.436} C_VEL
LIN {X 0,Y 363.843,Z 737.44,A -85,B 0,C 180,E1 11901.985,E2 11901.985} C_VEL
LIN {X 0,Y 363.594,Z 737.44,A -85,B 0,C 180,E1 11909.969,E2 11909.969} C_VEL
LIN {X 0,Y 363.353,Z 737.44,A -85,B 0,C 180,E1 11917.658,E2 11917.658} C_VEL
LIN {X 0,Y 363.385,Z 737.767,A -85,B 0,C 180,E1 11919.348,E2 11919.348} C_VEL
LIN {X 0,Y 365.678,Z 742.983,A -85,B 0,C 180,E1 11920.025,E2 11920.025} C_VEL
LIN {X 0,Y 368.473,Z 746.698,A -85,B 0,C 180,E1 11920.752,E2 11920.752} C_VEL
LIN {X 0,Y 382.929,Z 769.315,A -85,B 0,C 180,E1 11924.55,E2 11924.55} C_VEL
LIN {X 0,Y 396.796,Z 798.144,A -85,B 0,C 180,E1 11928.704,E2 11928.704} C_VEL
LIN {X 0,Y 405.536,Z 823.75,A -85,B 0,C 180,E1 11932.186,E2 11932.186} C_VEL
LIN {X 0,Y 398.839,Z 855.399,A -85,B 0,C 180,E1 11934.855,E2 11934.855} C_VEL
LIN {X 0,Y 391.131,Z 884.799,A -85,B 0,C 180,E1 11938.365,E2 11938.365} C_VEL
LIN {X 0,Y 383.369,Z 910.307,A -85,B 0,C 180,E1 11942.607,E2 11942.607} C_VEL
LIN {X 0,Y 376.535,Z 931.656,A -85,B 0,C 180,E1 11947.61,E2 11947.61} C_VEL
LIN {X 0,Y 371.291,Z 948.492,A -85,B 0,C 180,E1 11953.415,E2 11953.415} C_VEL
LIN {X 0,Y 368.356,Z 959.398,A -85,B 0,C 180,E1 11959.342,E2 11959.342} C_VEL
LIN {X 0,Y 367.039,Z 965.21,A -85,B 0,C 180,E1 11965.268,E2 11965.268} C_VEL
LIN {X 0,Y 367.036,Z 966.587,A -85,B 0,C 180,E1 11970,E2 11970} C_VEL
LIN {X 0,Y 367.054,Z 965.148,A -85,B 0,C 180,E1 11974.732,E2 11974.732} C_VEL
LIN {X 0,Y 368.363,Z 959.266,A -85,B 0,C 180,E1 11980.659,E2 11980.659} C_VEL
LIN {X 0,Y 371.646,Z 947.396,A -85,B 0,C 180,E1 11986.966,E2 11986.966} C_VEL
LIN {X 0,Y 376.702,Z 931.063,A -85,B 0,C 180,E1 11992.451,E2 11992.451} C_VEL
LIN {X 0,Y 383.654,Z 909.364,A -85,B 0,C 180,E1 11997.475,E2 11997.475} C_VEL
LIN {X 0,Y 391.341,Z 883.794,A -85,B 0,C 180,E1 12001.685,E2 12001.685} C_VEL
LIN {X 0,Y 399.325,Z 853.466,A -85,B 0,C 180,E1 12005.236,E2 12005.236} C_VEL
LIN {X 0,Y 405.401,Z 821.72,A -85,B 0,C 180,E1 12007.931,E2 12007.931} C_VEL
LIN {X 0,Y 393.257,Z 789.832,A -85,B 0,C 180,E1 12012.35,E2 12012.35} C_VEL
LIN {X 0,Y 378.079,Z 761.274,A -85,B 0,C 180,E1 12016.618,E2 12016.618} C_VEL
LIN {X 0,Y 366.223,Z 743.487,A -85,B 0,C 180,E1 12019.717,E2 12019.717} C_VEL
LIN {X 0,Y 363.506,Z 738.819,A -85,B 0,C 180,E1 12020.47,E2 12020.47} C_VEL
LIN {X 0,Y 363.398,Z 737.44,A -85,B 0,C 180,E1 12020.554,E2 12020.554} C_VEL
LIN {X 0,Y 363.411,Z 737.44,A -85,B 0,C 180,E1 12027.219,E2 12027.219} C_VEL
LIN {X 0,Y 363.615,Z 737.44,A -85,B 0,C 180,E1 12032.751,E2 12032.751} C_VEL
LIN {X 0,Y 363.869,Z 737.44,A -85,B 0,C 180,E1 12038.017,E2 12038.017} C_VEL
LIN {X 0,Y 364.316,Z 737.44,A -85,B 0,C 180,E1 12045.569,E2 12045.569} C_VEL
LIN {X 0,Y 364.663,Z 737.44,A -85,B 0,C 180,E1 12052.852,E2 12052.852} C_VEL
LIN {X 0,Y 365.015,Z 737.44,A -85,B 0,C 180,E1 12060.006,E2 12060.006} C_VEL
LIN {X 0,Y 364.659,Z 737.44,A -85,B 0,C 180,E1 12067.161,E2 12067.161} C_VEL
LIN {X 0,Y 364.18,Z 737.44,A -85,B 0,C 180,E1 12074.449,E2 12074.449} C_VEL
LIN {X 0,Y 363.833,Z 737.44,A -85,B 0,C 180,E1 12081.999,E2 12081.999} C_VEL
LIN {X 0,Y 363.63,Z 737.772,A -85,B 0,C 180,E1 12089.519,E2 12089.519} C_VEL
LIN {X 0,Y 365.96,Z 743.104,A -85,B 0,C 180,E1 12090.233,E2 12090.233} C_VEL
LIN {X 0,Y 368.869,Z 747.314,A -85,B 0,C 180,E1 12091.011,E2 12091.011} C_VEL
LIN {X 0,Y 386.279,Z 774.167,A -85,B 0,C 180,E1 12095.236,E2 12095.236} C_VEL
LIN {X 0,Y 403.181,Z 806.456,A -85,B 0,C 180,E1 12098.978,E2 12098.978} C_VEL
LIN {X 0,Y 411.496,Z 831.007,A -85,B 0,C 180,E1 12101.196,E2 12101.196} C_VEL
LIN {X 0,Y 405.487,Z 873.191,A -85,B 0,C 180,E1 12103.078,E2 12103.078} C_VEL
LIN {X 0,Y 398.033,Z 914.371,A -85,B 0,C 180,E1 12105.851,E2 12105.851} C_VEL
LIN {X 0,Y 389.799,Z 954.085,A -85,B 0,C 180,E1 12109.605,E2 12109.605} C_VEL
LIN {X 0,Y 381.729,Z 991.398,A -85,B 0,C 180,E1 12114.411,E2 12114.411} C_VEL
LIN {X 0,Y 375.288,Z 1021.908,A -85,B 0,C 180,E1 12119.607,E2 12119.607} C_VEL
LIN {X 0,Y 370.388,Z 1048.525,A -85,B 0,C 180,E1 12125.588,E2 12125.588} C_VEL
LIN {X 0,Y 367.496,Z 1068.931,A -85,B 0,C 180,E1 12131.774,E2 12131.774} C_VEL
LIN {X 0,Y 366.03,Z 1083.034,A -85,B 0,C 180,E1 12138.064,E2 12138.064} C_VEL
LIN {X 0,Y 365.625,Z 1090.465,A -85,B 0,C 180,E1 12143.63,E2 12143.63} C_VEL
LIN {X 0,Y 365.6,Z 1093.075,A -85,B 0,C 180,E1 12147.626,E2 12147.626} C_VEL
LIN {X 0,Y 365.502,Z 1093.2,A -85,B 0,C 180,E1 12151.626,E2 12151.626} C_VEL
LIN {X 0,Y 363.027,Z 1092.049,A -85,B 0,C 180,E1 12153.646,E2 12153.646} C_VEL
LIN {X 0,Y 357.855,Z 1088.597,A -85,B 0,C 180,E1 12157.021,E2 12157.021} C_VEL
LIN {X 0,Y 358.365,Z 1080.092,A -85,B 0,C 180,E1 12162.969,E2 12162.969} C_VEL
LIN {X 0,Y 359.803,Z 1066.45,A -85,B 0,C 180,E1 12168.909,E2 12168.909} C_VEL
LIN {X 0,Y 362.94,Z 1045.876,A -85,B 0,C 180,E1 12175.214,E2 12175.214} C_VEL
LIN {X 0,Y 368.305,Z 1018.951,A -85,B 0,C 180,E1 12181.298,E2 12181.298} C_VEL
LIN {X 0,Y 375.514,Z 986.293,A -85,B 0,C 180,E1 12186.839,E2 12186.839} C_VEL
LIN {X 0,Y 383.503,Z 951.429,A -85,B 0,C 180,E1 12191.3,E2 12191.3} C_VEL
LIN {X 0,Y 392.079,Z 912.266,A -85,B 0,C 180,E1 12195.001,E2 12195.001} C_VEL
LIN {X 0,Y 399.831,Z 871.13,A -85,B 0,C 180,E1 12197.765,E2 12197.765} C_VEL
LIN {X 0,Y 405.205,Z 831.832,A -85,B 0,C 180,E1 12199.602,E2 12199.602} C_VEL
LIN {X 0,Y 395.038,Z 804.021,A -85,B 0,C 180,E1 12202.349,E2 12202.349} C_VEL
LIN {X 0,Y 377.736,Z 772.574,A -85,B 0,C 180,E1 12206.381,E2 12206.381} C_VEL
LIN {X 0,Y 362.023,Z 748.775,A -85,B 0,C 180,E1 12210.471,E2 12210.471} C_VEL
LIN {X 0,Y 358.559,Z 743.527,A -85,B 0,C 180,E1 12211.479,E2 12211.479} C_VEL
LIN {X 0,Y 355.805,Z 738.548,A -85,B 0,C 180,E1 12212.347,E2 12212.347} C_VEL
LIN {X 0,Y 355.725,Z 737.44,A -85,B 0,C 180,E1 12212.427,E2 12212.427} C_VEL
LIN {X 0,Y 356.049,Z 737.44,A -85,B 0,C 180,E1 12220.107,E2 12220.107} C_VEL
LIN {X 0,Y 356.325,Z 737.44,A -85,B 0,C 180,E1 12227.754,E2 12227.754} C_VEL
LIN {X 0,Y 356.811,Z 737.44,A -85,B 0,C 180,E1 12235.126,E2 12235.126} C_VEL
LIN {X 0,Y 357.113,Z 737.44,A -85,B 0,C 180,E1 12239.994,E2 12239.994} C_VEL
LIN {X 0,Y 356.713,Z 737.44,A -85,B 0,C 180,E1 12247.308,E2 12247.308} C_VEL
LIN {X 0,Y 356.242,Z 737.44,A -85,B 0,C 180,E1 12254.765,E2 12254.765} C_VEL
LIN {X 0,Y 355.891,Z 737.44,A -85,B 0,C 180,E1 12262.503,E2 12262.503} C_VEL
LIN {X 0,Y 355.712,Z 737.44,A -85,B 0,C 180,E1 12267.907,E2 12267.907} C_VEL
LIN {X 0,Y 355.445,Z 737.44,A -85,B 0,C 180,E1 12275.974,E2 12275.974} C_VEL
LIN {X 0,Y 355.439,Z 737.478,A -85,B 0,C 180,E1 12277.423,E2 12277.423} C_VEL
LIN {X 0,Y 357.547,Z 742.813,A -85,B 0,C 180,E1 12278.122,E2 12278.122} C_VEL
LIN {X 0,Y 360.562,Z 746.51,A -85,B 0,C 180,E1 12278.962,E2 12278.962} C_VEL
LIN {X 0,Y 375.63,Z 769.659,A -85,B 0,C 180,E1 12283.175,E2 12283.175} C_VEL
LIN {X 0,Y 388.863,Z 796.349,A -85,B 0,C 180,E1 12287.283,E2 12287.283} C_VEL
LIN {X 0,Y 399.383,Z 825.778,A -85,B 0,C 180,E1 12291.498,E2 12291.498} C_VEL
LIN {X 0,Y 392.325,Z 858.157,A -85,B 0,C 180,E1 12294.318,E2 12294.318} C_VEL
LIN {X 0,Y 384.583,Z 886.368,A -85,B 0,C 180,E1 12297.762,E2 12297.762} C_VEL
LIN {X 0,Y 376.647,Z 911.324,A -85,B 0,C 180,E1 12301.972,E2 12301.972} C_VEL
LIN {X 0,Y 369.351,Z 933.087,A -85,B 0,C 180,E1 12307.151,E2 12307.151} C_VEL
LIN {X 0,Y 363.759,Z 950.077,A -85,B 0,C 180,E1 12313.154,E2 12313.154} C_VEL
LIN {X 0,Y 360.691,Z 960.763,A -85,B 0,C 180,E1 12319.112,E2 12319.112} C_VEL
LIN {X 0,Y 359.269,Z 966.563,A -85,B 0,C 180,E1 12325.165,E2 12325.165} C_VEL
LIN {X 0,Y 359.251,Z 967.935,A -85,B 0,C 180,E1 12330,E2 12330} C_VEL
LIN {X 0,Y 359.286,Z 966.502,A -85,B 0,C 180,E1 12334.835,E2 12334.835} C_VEL
LIN {X 0,Y 360.698,Z 960.633,A -85,B 0,C 180,E1 12340.888,E2 12340.888} C_VEL
LIN {X 0,Y 363.889,Z 949.66,A -85,B 0,C 180,E1 12346.932,E2 12346.932} C_VEL
LIN {X 0,Y 369.506,Z 932.502,A -85,B 0,C 180,E1 12352.913,E2 12352.913} C_VEL
LIN {X 0,Y 376.85,Z 910.683,A -85,B 0,C 180,E1 12358.052,E2 12358.052} C_VEL
LIN {X 0,Y 384.779,Z 885.373,A -85,B 0,C 180,E1 12362.29,E2 12362.29} C_VEL
LIN {X 0,Y 392.841,Z 856.164,A -85,B 0,C 180,E1 12365.78,E2 12365.78} C_VEL
LIN {X 0,Y 399.139,Z 824.964,A -85,B 0,C 180,E1 12368.516,E2 12368.516} C_VEL
LIN {X 0,Y 388.616,Z 795.966,A -85,B 0,C 180,E1 12372.678,E2 12372.678} C_VEL
LIN {X 0,Y 374.318,Z 767.503,A -85,B 0,C 180,E1 12377.076,E2 12377.076} C_VEL
LIN {X 0,Y 361.779,Z 748.588,A -85,B 0,C 180,E1 12380.553,E2 12380.553} C_VEL
LIN {X 0,Y 358.36,Z 743.563,A -85,B 0,C 180,E1 12381.53,E2 12381.53} C_VEL
LIN {X 0,Y 355.535,Z 738.373,A -85,B 0,C 180,E1 12382.396,E2 12382.396} C_VEL
LIN {X 0,Y 355.435,Z 737.44,A -85,B 0,C 180,E1 12382.895,E2 12382.895} C_VEL
LIN {X 0,Y 355.543,Z 737.44,A -85,B 0,C 180,E1 12389.28,E2 12389.28} C_VEL
LIN {X 0,Y 355.752,Z 737.44,A -85,B 0,C 180,E1 12394.822,E2 12394.822} C_VEL
LIN {X 0,Y 356.268,Z 737.44,A -85,B 0,C 180,E1 12402.702,E2 12402.702} C_VEL
LIN {X 0,Y 356.57,Z 737.44,A -85,B 0,C 180,E1 12410.229,E2 12410.229} C_VEL
LIN {X 0,Y 356.98,Z 737.44,A -85,B 0,C 180,E1 12417.576,E2 12417.576} C_VEL
LIN {X 0,Y 357.071,Z 737.44,A -85,B 0,C 180,E1 12422.436,E2 12422.436} C_VEL
LIN {X 0,Y 356.493,Z 737.44,A -85,B 0,C 180,E1 12429.786,E2 12429.786} C_VEL
LIN {X 0,Y 356.152,Z 737.44,A -85,B 0,C 180,E1 12437.317,E2 12437.317} C_VEL
LIN {X 0,Y 355.761,Z 737.44,A -85,B 0,C 180,E1 12445.191,E2 12445.191} C_VEL
LIN {X 0,Y 355.747,Z 738.233,A -85,B 0,C 180,E1 12447.657,E2 12447.657} C_VEL
LIN {X 0,Y 358.481,Z 743.461,A -85,B 0,C 180,E1 12448.528,E2 12448.528} C_VEL
LIN {X 0,Y 373.187,Z 765.418,A -85,B 0,C 180,E1 12452.521,E2 12452.521} C_VEL
LIN {X 0,Y 389.674,Z 793.368,A -85,B 0,C 180,E1 12456.425,E2 12456.425} C_VEL
LIN {X 0,Y 401.555,Z 820.398,A -85,B 0,C 180,E1 12459.341,E2 12459.341} C_VEL
LIN {X 0,Y 405.323,Z 834.287,A -85,B 0,C 180,E1 12460.554,E2 12460.554} C_VEL
LIN {X 0,Y 398.821,Z 876.755,A -85,B 0,C 180,E1 12462.549,E2 12462.549} C_VEL
LIN {X 0,Y 390.577,Z 919.109,A -85,B 0,C 180,E1 12465.56,E2 12465.56} C_VEL
LIN {X 0,Y 382.282,Z 956.975,A -85,B 0,C 180,E1 12469.338,E2 12469.338} C_VEL
LIN {X 0,Y 374.344,Z 991.75,A -85,B 0,C 180,E1 12473.99,E2 12473.99} C_VEL
LIN {X 0,Y 367.636,Z 1021.907,A -85,B 0,C 180,E1 12479.295,E2 12479.295} C_VEL
LIN {X 0,Y 362.639,Z 1047.862,A -85,B 0,C 180,E1 12485.323,E2 12485.323} C_VEL
LIN {X 0,Y 359.712,Z 1067.599,A -85,B 0,C 180,E1 12491.499,E2 12491.499} C_VEL
LIN {X 0,Y 358.247,Z 1081.525,A -85,B 0,C 180,E1 12497.801,E2 12497.801} C_VEL
LIN {X 0,Y 357.841,Z 1089.138,A -85,B 0,C 180,E1 12503.561,E2 12503.561} C_VEL
LIN {X 0,Y 357.802,Z 1091.717,A -85,B 0,C 180,E1 12507.575,E2 12507.575} C_VEL
LIN {X 0,Y 357.727,Z 1091.704,A -85,B 0,C 180,E1 12512.425,E2 12512.425} C_VEL
LIN {X 0,Y 357.855,Z 1088.597,A -85,B 0,C 180,E1 12517.021,E2 12517.021} C_VEL
LIN {X 0,Y 355.49,Z 1085.998,A -85,B 0,C 180,E1 12519.05,E2 12519.05} C_VEL
LIN {X 0,Y 350.485,Z 1080.758,A -85,B 0,C 180,E1 12522.063,E2 12522.063} C_VEL
LIN {X 0,Y 350.443,Z 1080.118,A -85,B 0,C 180,E1 12522.41,E2 12522.41} C_VEL
LIN {X 0,Y 351.874,Z 1066.33,A -85,B 0,C 180,E1 12528.806,E2 12528.806} C_VEL
LIN {X 0,Y 355.017,Z 1046.229,A -85,B 0,C 180,E1 12535.243,E2 12535.243} C_VEL
LIN {X 0,Y 360.692,Z 1019.019,A -85,B 0,C 180,E1 12541.647,E2 12541.647} C_VEL
LIN {X 0,Y 368.23,Z 986.691,A -85,B 0,C 180,E1 12547.311,E2 12547.311} C_VEL
LIN {X 0,Y 376.736,Z 951.491,A -85,B 0,C 180,E1 12551.932,E2 12551.932} C_VEL
LIN {X 0,Y 385.706,Z 912.492,A -85,B 0,C 180,E1 12555.695,E2 12555.695} C_VEL
LIN {X 0,Y 393.892,Z 870.743,A -85,B 0,C 180,E1 12558.548,E2 12558.548} C_VEL
LIN {X 0,Y 399.207,Z 834.549,A -85,B 0,C 180,E1 12560.271,E2 12560.271} C_VEL
LIN {X 0,Y 389.83,Z 808.222,A -85,B 0,C 180,E1 12562.985,E2 12562.985} C_VEL
LIN {X 0,Y 373.58,Z 778.047,A -85,B 0,C 180,E1 12567,E2 12567} C_VEL
LIN {X 0,Y 355.94,Z 750.636,A -85,B 0,C 180,E1 12571.839,E2 12571.839} C_VEL
LIN {X 0,Y 350.619,Z 743.45,A -85,B 0,C 180,E1 12573.489,E2 12573.489} C_VEL
LIN {X 0,Y 347.893,Z 738.195,A -85,B 0,C 180,E1 12574.447,E2 12574.447} C_VEL
LIN {X 0,Y 348.105,Z 737.44,A -85,B 0,C 180,E1 12579.634,E2 12579.634} C_VEL
LIN {X 0,Y 348.366,Z 737.44,A -85,B 0,C 180,E1 12587.444,E2 12587.444} C_VEL
LIN {X 0,Y 348.913,Z 737.44,A -85,B 0,C 180,E1 12595.015,E2 12595.015} C_VEL
LIN {X 0,Y 349.211,Z 737.44,A -85,B 0,C 180,E1 12599.994,E2 12599.994} C_VEL
LIN {X 0,Y 348.778,Z 737.44,A -85,B 0,C 180,E1 12607.475,E2 12607.475} C_VEL
LIN {X 0,Y 348.293,Z 737.44,A -85,B 0,C 180,E1 12615.11,E2 12615.11} C_VEL
LIN {X 0,Y 348.091,Z 737.44,A -85,B 0,C 180,E1 12620.353,E2 12620.353} C_VEL
LIN {X 0,Y 347.694,Z 737.44,A -85,B 0,C 180,E1 12628.609,E2 12628.609} C_VEL
LIN {X 0,Y 347.515,Z 737.44,A -85,B 0,C 180,E1 12635.286,E2 12635.286} C_VEL
LIN {X 0,Y 349.581,Z 742.703,A -85,B 0,C 180,E1 12636.068,E2 12636.068} C_VEL
LIN {X 0,Y 352.703,Z 746.399,A -85,B 0,C 180,E1 12637.023,E2 12637.023} C_VEL
LIN {X 0,Y 368.556,Z 770.31,A -85,B 0,C 180,E1 12641.767,E2 12641.767} C_VEL
LIN {X 0,Y 381.506,Z 796.072,A -85,B 0,C 180,E1 12645.982,E2 12645.982} C_VEL
LIN {X 0,Y 391.998,Z 825.221,A -85,B 0,C 180,E1 12650.319,E2 12650.319} C_VEL
LIN {X 0,Y 393.016,Z 830.455,A -85,B 0,C 180,E1 12651.023,E2 12651.023} C_VEL
LIN {X 0,Y 385.141,Z 863.602,A -85,B 0,C 180,E1 12654.042,E2 12654.042} C_VEL
LIN {X 0,Y 376.548,Z 892.854,A -85,B 0,C 180,E1 12657.876,E2 12657.876} C_VEL
LIN {X 0,Y 368.242,Z 917.306,A -85,B 0,C 180,E1 12662.354,E2 12662.354} C_VEL
LIN {X 0,Y 361.213,Z 936.966,A -85,B 0,C 180,E1 12667.422,E2 12667.422} C_VEL
LIN {X 0,Y 355.952,Z 952.412,A -85,B 0,C 180,E1 12673.223,E2 12673.223} C_VEL
LIN {X 0,Y 353.042,Z 962.125,A -85,B 0,C 180,E1 12678.874,E2 12678.874} C_VEL
LIN {X 0,Y 351.514,Z 967.914,A -85,B 0,C 180,E1 12685.059,E2 12685.059} C_VEL
LIN {X 0,Y 351.492,Z 969.279,A -85,B 0,C 180,E1 12690,E2 12690} C_VEL
LIN {X 0,Y 351.532,Z 967.853,A -85,B 0,C 180,E1 12694.942,E2 12694.942} C_VEL
LIN {X 0,Y 353.049,Z 961.996,A -85,B 0,C 180,E1 12701.127,E2 12701.127} C_VEL
LIN {X 0,Y 356.408,Z 951.048,A -85,B 0,C 180,E1 12707.299,E2 12707.299} C_VEL
LIN {X 0,Y 361.931,Z 935.077,A -85,B 0,C 180,E1 12713.06,E2 12713.06} C_VEL
LIN {X 0,Y 369.524,Z 913.592,A -85,B 0,C 180,E1 12718.335,E2 12718.335} C_VEL
LIN {X 0,Y 377.825,Z 888.317,A -85,B 0,C 180,E1 12722.72,E2 12722.72} C_VEL
LIN {X 0,Y 386.157,Z 859.681,A -85,B 0,C 180,E1 12726.26,E2 12726.26} C_VEL
LIN {X 0,Y 393.094,Z 829.466,A -85,B 0,C 180,E1 12728.962,E2 12728.962} C_VEL
LIN {X 0,Y 383.774,Z 801.588,A -85,B 0,C 180,E1 12733.087,E2 12733.087} C_VEL
LIN {X 0,Y 370.236,Z 773.425,A -85,B 0,C 180,E1 12737.578,E2 12737.578} C_VEL
LIN {X 0,Y 355.353,Z 750.235,A -85,B 0,C 180,E1 12742.031,E2 12742.031} C_VEL
LIN {X 0,Y 350.684,Z 743.77,A -85,B 0,C 180,E1 12743.465,E2 12743.465} C_VEL
LIN {X 0,Y 347.569,Z 738.509,A -85,B 0,C 180,E1 12744.503,E2 12744.503} C_VEL
LIN {X 0,Y 347.49,Z 737.44,A -85,B 0,C 180,E1 12744.64,E2 12744.64} C_VEL
LIN {X 0,Y 347.682,Z 737.44,A -85,B 0,C 180,E1 12751.39,E2 12751.39} C_VEL
LIN {X 0,Y 348.133,Z 737.44,A -85,B 0,C 180,E1 12759.649,E2 12759.649} C_VEL
LIN {X 0,Y 348.406,Z 737.44,A -85,B 0,C 180,E1 12764.895,E2 12764.895} C_VEL
LIN {X 0,Y 348.797,Z 737.44,A -85,B 0,C 180,E1 12772.525,E2 12772.525} C_VEL
LIN {X 0,Y 349.223,Z 737.44,A -85,B 0,C 180,E1 12780.006,E2 12780.006} C_VEL
LIN {X 0,Y 348.784,Z 737.44,A -85,B 0,C 180,E1 12787.488,E2 12787.488} C_VEL
LIN {X 0,Y 348.277,Z 737.44,A -85,B 0,C 180,E1 12795.124,E2 12795.124} C_VEL
LIN {X 0,Y 347.895,Z 737.44,A -85,B 0,C 180,E1 12803.063,E2 12803.063} C_VEL
LIN {X 0,Y 347.852,Z 737.635,A -85,B 0,C 180,E1 12805.554,E2 12805.554} C_VEL
LIN {X 0,Y 350.036,Z 742.914,A -85,B 0,C 180,E1 12806.372,E2 12806.372} C_VEL
LIN {X 0,Y 352.926,Z 746.554,A -85,B 0,C 180,E1 12807.275,E2 12807.275} C_VEL
LIN {X 0,Y 368.64,Z 769.915,A -85,B 0,C 180,E1 12811.754,E2 12811.754} C_VEL
LIN {X 0,Y 385.468,Z 799.2,A -85,B 0,C 180,E1 12815.927,E2 12815.927} C_VEL
LIN {X 0,Y 396.38,Z 825.292,A -85,B 0,C 180,E1 12818.844,E2 12818.844} C_VEL
LIN {X 0,Y 399.275,Z 836.387,A -85,B 0,C 180,E1 12819.856,E2 12819.856} C_VEL
LIN {X 0,Y 392.606,Z 877.759,A -85,B 0,C 180,E1 12821.863,E2 12821.863} C_VEL
LIN {X 0,Y 384.249,Z 918.714,A -85,B 0,C 180,E1 12824.828,E2 12824.828} C_VEL
LIN {X 0,Y 375.446,Z 956.865,A -85,B 0,C 180,E1 12828.705,E2 12828.705} C_VEL
LIN {X 0,Y 367.26,Z 990.872,A -85,B 0,C 180,E1 12833.35,E2 12833.35} C_VEL
LIN {X 0,Y 360.337,Z 1020.521,A -85,B 0,C 180,E1 12838.671,E2 12838.671} C_VEL
LIN {X 0,Y 355.001,Z 1046.23,A -85,B 0,C 180,E1 12844.756,E2 12844.756} C_VEL
LIN {X 0,Y 351.923,Z 1066.274,A -85,B 0,C 180,E1 12851.171,E2 12851.171} C_VEL
LIN {X 0,Y 350.468,Z 1080.012,A -85,B 0,C 180,E1 12857.526,E2 12857.526} C_VEL
LIN {X 0,Y 350.089,Z 1086.937,A -85,B 0,C 180,E1 12862.545,E2 12862.545} C_VEL
LIN {X 0,Y 350.01,Z 1090.36,A -85,B 0,C 180,E1 12867.521,E2 12867.521} C_VEL
LIN {X 0,Y 349.937,Z 1090.347,A -85,B 0,C 180,E1 12872.479,E2 12872.479} C_VEL
LIN {X 0,Y 350.088,Z 1086.935,A -85,B 0,C 180,E1 12877.454,E2 12877.454} C_VEL
LIN {X 0,Y 350.443,Z 1080.118,A -85,B 0,C 180,E1 12882.41,E2 12882.41} C_VEL
LIN {X 0,Y 348.278,Z 1076.157,A -85,B 0,C 180,E1 12884.432,E2 12884.432} C_VEL
LIN {X 0,Y 343.661,Z 1069.218,A -85,B 0,C 180,E1 12887.43,E2 12887.43} C_VEL
LIN {X 0,Y 343.663,Z 1068.38,A -85,B 0,C 180,E1 12887.771,E2 12887.771} C_VEL
LIN {X 0,Y 346.43,Z 1050.296,A -85,B 0,C 180,E1 12894.187,E2 12894.187} C_VEL
LIN {X 0,Y 351.681,Z 1025,A -85,B 0,C 180,E1 12900.721,E2 12900.721} C_VEL
LIN {X 0,Y 359.127,Z 994.714,A -85,B 0,C 180,E1 12906.548,E2 12906.548} C_VEL
LIN {X 0,Y 367.609,Z 961.112,A -85,B 0,C 180,E1 12911.426,E2 12911.426} C_VEL
LIN {X 0,Y 376.973,Z 922.768,A -85,B 0,C 180,E1 12915.541,E2 12915.541} C_VEL
LIN {X 0,Y 385.8,Z 882.681,A -85,B 0,C 180,E1 12918.598,E2 12918.598} C_VEL
LIN {X 0,Y 392.781,Z 843.426,A -85,B 0,C 180,E1 12920.65,E2 12920.65} C_VEL
LIN {X 0,Y 392.978,Z 836.463,A -85,B 0,C 180,E1 12921.043,E2 12921.043} C_VEL
LIN {X 0,Y 384.51,Z 811.997,A -85,B 0,C 180,E1 12923.685,E2 12923.685} C_VEL
LIN {X 0,Y 368.993,Z 782.62,A -85,B 0,C 180,E1 12927.761,E2 12927.761} C_VEL
LIN {X 0,Y 352.381,Z 756.806,A -85,B 0,C 180,E1 12932.487,E2 12932.487} C_VEL
LIN {X 0,Y 343.216,Z 743.8,A -85,B 0,C 180,E1 12935.543,E2 12935.543} C_VEL
LIN {X 0,Y 340.24,Z 739.345,A -85,B 0,C 180,E1 12936.647,E2 12936.647} C_VEL
LIN {X 0,Y 340.046,Z 737.44,A -85,B 0,C 180,E1 12936.893,E2 12936.893} C_VEL
LIN {X 0,Y 340.311,Z 737.44,A -85,B 0,C 180,E1 12944.513,E2 12944.513} C_VEL
LIN {X 0,Y 340.829,Z 737.44,A -85,B 0,C 180,E1 12952.336,E2 12952.336} C_VEL
LIN {X 0,Y 341.323,Z 737.44,A -85,B 0,C 180,E1 12959.993,E2 12959.993} C_VEL
LIN {X 0,Y 340.838,Z 737.44,A -85,B 0,C 180,E1 12967.651,E2 12967.651} C_VEL
LIN {X 0,Y 340.359,Z 737.44,A -85,B 0,C 180,E1 12975.471,E2 12975.471} C_VEL
LIN {X 0,Y 340.117,Z 737.44,A -85,B 0,C 180,E1 12980.853,E2 12980.853} C_VEL
LIN {X 0,Y 339.759,Z 737.44,A -85,B 0,C 180,E1 12989.341,E2 12989.341} C_VEL
LIN {X 0,Y 339.612,Z 738.034,A -85,B 0,C 180,E1 12992.979,E2 12992.979} C_VEL
LIN {X 0,Y 342.037,Z 743.14,A -85,B 0,C 180,E1 12993.932,E2 12993.932} C_VEL
LIN {X 0,Y 344.869,Z 746.273,A -85,B 0,C 180,E1 12994.884,E2 12994.884} C_VEL
LIN {X 0,Y 359.248,Z 767.579,A -85,B 0,C 180,E1 12999.568,E2 12999.568} C_VEL
LIN {X 0,Y 372.78,Z 792.396,A -85,B 0,C 180,E1 13004.055,E2 13004.055} C_VEL
LIN {X 0,Y 383.681,Z 821.012,A -85,B 0,C 180,E1 13008.553,E2 13008.553} C_VEL
LIN {X 0,Y 386.881,Z 833.458,A -85,B 0,C 180,E1 13010.388,E2 13010.388} C_VEL
LIN {X 0,Y 378.555,Z 866.466,A -85,B 0,C 180,E1 13013.494,E2 13013.494} C_VEL
LIN {X 0,Y 369.632,Z 895.448,A -85,B 0,C 180,E1 13017.41,E2 13017.41} C_VEL
LIN {X 0,Y 360.78,Z 920.355,A -85,B 0,C 180,E1 13022.141,E2 13022.141} C_VEL
LIN {X 0,Y 353.581,Z 939.616,A -85,B 0,C 180,E1 13027.334,E2 13027.334} C_VEL
LIN {X 0,Y 348.149,Z 954.76,A -85,B 0,C 180,E1 13033.303,E2 13033.303} C_VEL
LIN {X 0,Y 344.929,Z 965.059,A -85,B 0,C 180,E1 13039.888,E2 13039.888} C_VEL
LIN {X 0,Y 343.674,Z 970.285,A -85,B 0,C 180,E1 13047.475,E2 13047.475} C_VEL
LIN {X 0,Y 343.677,Z 970.25,A -85,B 0,C 180,E1 13052.525,E2 13052.525} C_VEL
LIN {X 0,Y 344.638,Z 966.078,A -85,B 0,C 180,E1 13059.034,E2 13059.034} C_VEL
LIN {X 0,Y 347.234,Z 957.467,A -85,B 0,C 180,E1 13065.166,E2 13065.166} C_VEL
LIN {X 0,Y 352.343,Z 943.007,A -85,B 0,C 180,E1 13071.422,E2 13071.422} C_VEL
LIN {X 0,Y 359.967,Z 922.712,A -85,B 0,C 180,E1 13077.219,E2 13077.219} C_VEL
LIN {X 0,Y 368.408,Z 898.848,A -85,B 0,C 180,E1 13081.945,E2 13081.945} C_VEL
LIN {X 0,Y 377.336,Z 870.519,A -85,B 0,C 180,E1 13085.93,E2 13085.93} C_VEL
LIN {X 0,Y 385.568,Z 839.01,A -85,B 0,C 180,E1 13089.058,E2 13089.058} C_VEL
LIN {X 0,Y 386.666,Z 831.153,A -85,B 0,C 180,E1 13089.785,E2 13089.785} C_VEL
LIN {X 0,Y 376.836,Z 802.07,A -85,B 0,C 180,E1 13094.288,E2 13094.288} C_VEL
LIN {X 0,Y 363.309,Z 774.172,A -85,B 0,C 180,E1 13099.012,E2 13099.012} C_VEL
LIN {X 0,Y 347.958,Z 750.656,A -85,B 0,C 180,E1 13103.943,E2 13103.943} C_VEL
LIN {X 0,Y 342.993,Z 743.932,A -85,B 0,C 180,E1 13105.614,E2 13105.614} C_VEL
LIN {X 0,Y 339.748,Z 739.043,A -85,B 0,C 180,E1 13106.795,E2 13106.795} C_VEL
LIN {X 0,Y 339.585,Z 737.44,A -85,B 0,C 180,E1 13107.021,E2 13107.021} C_VEL
LIN {X 0,Y 339.802,Z 737.44,A -85,B 0,C 180,E1 13113.551,E2 13113.551} C_VEL
LIN {X 0,Y 340.325,Z 737.44,A -85,B 0,C 180,E1 13121.865,E2 13121.865} C_VEL
LIN {X 0,Y 340.725,Z 737.44,A -85,B 0,C 180,E1 13129.77,E2 13129.77} C_VEL
LIN {X 0,Y 341.17,Z 737.44,A -85,B 0,C 180,E1 13137.463,E2 13137.463} C_VEL
LIN {X 0,Y 341.245,Z 737.44,A -85,B 0,C 180,E1 13142.549,E2 13142.549} C_VEL
LIN {X 0,Y 340.611,Z 737.44,A -85,B 0,C 180,E1 13150.247,E2 13150.247} C_VEL
LIN {X 0,Y 340.223,Z 737.44,A -85,B 0,C 180,E1 13158.155,E2 13158.155} C_VEL
LIN {X 0,Y 339.979,Z 737.44,A -85,B 0,C 180,E1 13163.198,E2 13163.198} C_VEL
LIN {X 0,Y 342.107,Z 742.888,A -85,B 0,C 180,E1 13164.132,E2 13164.132} C_VEL
LIN {X 0,Y 345.058,Z 746.157,A -85,B 0,C 180,E1 13165.135,E2 13165.135} C_VEL
LIN {X 0,Y 361.569,Z 770.545,A -85,B 0,C 180,E1 13170.255,E2 13170.255} C_VEL
LIN {X 0,Y 378.59,Z 799.715,A -85,B 0,C 180,E1 13174.745,E2 13174.745} C_VEL
LIN {X 0,Y 390.062,Z 826.525,A -85,B 0,C 180,E1 13177.963,E2 13177.963} C_VEL
LIN {X 0,Y 393.329,Z 838.28,A -85,B 0,C 180,E1 13179.129,E2 13179.129} C_VEL
LIN {X 0,Y 386.277,Z 879.545,A -85,B 0,C 180,E1 13181.199,E2 13181.199} C_VEL
LIN {X 0,Y 378.041,Z 918.258,A -85,B 0,C 180,E1 13184.068,E2 13184.068} C_VEL
LIN {X 0,Y 369.145,Z 954.978,A -85,B 0,C 180,E1 13187.833,E2 13187.833} C_VEL
LIN {X 0,Y 360.508,Z 988.909,A -85,B 0,C 180,E1 13192.504,E2 13192.504} C_VEL
LIN {X 0,Y 353.145,Z 1018.867,A -85,B 0,C 180,E1 13197.958,E2 13197.958} C_VEL
LIN {X 0,Y 347.457,Z 1044.643,A -85,B 0,C 180,E1 13204.168,E2 13204.168} C_VEL
LIN {X 0,Y 344.133,Z 1064.744,A -85,B 0,C 180,E1 13210.728,E2 13210.728} C_VEL
LIN {X 0,Y 342.687,Z 1078.556,A -85,B 0,C 180,E1 13217.238,E2 13217.238} C_VEL
LIN {X 0,Y 342.271,Z 1085.527,A -85,B 0,C 180,E1 13222.374,E2 13222.374} C_VEL
LIN {X 0,Y 342.227,Z 1089.004,A -85,B 0,C 180,E1 13227.464,E2 13227.464} C_VEL
LIN {X 0,Y 342.159,Z 1088.992,A -85,B 0,C 180,E1 13232.536,E2 13232.536} C_VEL
LIN {X 0,Y 342.271,Z 1085.527,A -85,B 0,C 180,E1 13237.626,E2 13237.626} C_VEL
LIN {X 0,Y 342.812,Z 1076.928,A -85,B 0,C 180,E1 13243.678,E2 13243.678} C_VEL
LIN {X 0,Y 343.663,Z 1068.38,A -85,B 0,C 180,E1 13247.771,E2 13247.771} C_VEL
LIN {X 0,Y 340.722,Z 1061.525,A -85,B 0,C 180,E1 13250.424,E2 13250.424} C_VEL
LIN {X 0,Y 337.924,Z 1053.959,A -85,B 0,C 180,E1 13253.073,E2 13253.073} C_VEL
LIN {X 0,Y 342.588,Z 1031.052,A -85,B 0,C 180,E1 13259.619,E2 13259.619} C_VEL
LIN {X 0,Y 349.358,Z 1003.996,A -85,B 0,C 180,E1 13265.424,E2 13265.424} C_VEL
LIN {X 0,Y 358.049,Z 971.736,A -85,B 0,C 180,E1 13270.652,E2 13270.652} C_VEL
LIN {X 0,Y 367.693,Z 934.991,A -85,B 0,C 180,E1 13275.083,E2 13275.083} C_VEL
LIN {X 0,Y 377.059,Z 895.863,A -85,B 0,C 180,E1 13278.49,E2 13278.49} C_VEL
LIN {X 0,Y 385.046,Z 855.526,A -85,B 0,C 180,E1 13280.931,E2 13280.931} C_VEL
LIN {X 0,Y 387.179,Z 839.416,A -85,B 0,C 180,E1 13281.722,E2 13281.722} C_VEL
LIN {X 0,Y 379.247,Z 816.163,A -85,B 0,C 180,E1 13284.37,E2 13284.37} C_VEL
LIN {X 0,Y 365.096,Z 788.401,A -85,B 0,C 180,E1 13288.339,E2 13288.339} C_VEL
LIN {X 0,Y 348.885,Z 762.826,A -85,B 0,C 180,E1 13293.15,E2 13293.15} C_VEL
LIN {X 0,Y 339.851,Z 750.101,A -85,B 0,C 180,E1 13296.271,E2 13296.271} C_VEL
LIN {X 0,Y 335.878,Z 744.164,A -85,B 0,C 180,E1 13297.815,E2 13297.815} C_VEL
LIN {X 0,Y 332.546,Z 739.591,A -85,B 0,C 180,E1 13299.193,E2 13299.193} C_VEL
LIN {X 0,Y 332.231,Z 737.44,A -85,B 0,C 180,E1 13299.544,E2 13299.544} C_VEL
LIN {X 0,Y 332.466,Z 737.44,A -85,B 0,C 180,E1 13306.833,E2 13306.833} C_VEL
LIN {X 0,Y 333.063,Z 737.44,A -85,B 0,C 180,E1 13314.777,E2 13314.777} C_VEL
LIN {X 0,Y 333.252,Z 737.44,A -85,B 0,C 180,E1 13321.86,E2 13321.86} C_VEL
LIN {X 0,Y 332.908,Z 737.44,A -85,B 0,C 180,E1 13327.834,E2 13327.834} C_VEL
LIN {X 0,Y 332.4,Z 737.44,A -85,B 0,C 180,E1 13335.851,E2 13335.851} C_VEL
LIN {X 0,Y 332.12,Z 737.44,A -85,B 0,C 180,E1 13341.379,E2 13341.379} C_VEL
LIN {X 0,Y 331.801,Z 737.44,A -85,B 0,C 180,E1 13349.893,E2 13349.893} C_VEL
LIN {X 0,Y 331.824,Z 738.6,A -85,B 0,C 180,E1 13350.37,E2 13350.37} C_VEL
LIN {X 0,Y 334.689,Z 743.62,A -85,B 0,C 180,E1 13351.601,E2 13351.601} C_VEL
LIN {X 0,Y 337.073,Z 746.183,A -85,B 0,C 180,E1 13352.5,E2 13352.5} C_VEL
LIN {X 0,Y 350.703,Z 765.843,A -85,B 0,C 180,E1 13357.374,E2 13357.374} C_VEL
LIN {X 0,Y 363.882,Z 789.12,A -85,B 0,C 180,E1 13362.002,E2 13362.002} C_VEL
LIN {X 0,Y 374.751,Z 815.054,A -85,B 0,C 180,E1 13366.385,E2 13366.385} C_VEL
LIN {X 0,Y 380.817,Z 836.101,A -85,B 0,C 180,E1 13369.71,E2 13369.71} C_VEL
LIN {X 0,Y 372.393,Z 868.095,A -85,B 0,C 180,E1 13372.789,E2 13372.789} C_VEL
LIN {X 0,Y 363.483,Z 895.969,A -85,B 0,C 180,E1 13376.589,E2 13376.589} C_VEL
LIN {X 0,Y 354.479,Z 920.353,A -85,B 0,C 180,E1 13381.223,E2 13381.223} C_VEL
LIN {X 0,Y 346.38,Z 941.025,A -85,B 0,C 180,E1 13386.835,E2 13386.835} C_VEL
LIN {X 0,Y 340.673,Z 956.141,A -85,B 0,C 180,E1 13392.925,E2 13392.925} C_VEL
LIN {X 0,Y 337.248,Z 966.416,A -85,B 0,C 180,E1 13399.655,E2 13399.655} C_VEL
LIN {X 0,Y 335.91,Z 971.631,A -85,B 0,C 180,E1 13407.417,E2 13407.417} C_VEL
LIN {X 0,Y 335.914,Z 971.597,A -85,B 0,C 180,E1 13412.583,E2 13412.583} C_VEL
LIN {X 0,Y 336.74,Z 968.165,A -85,B 0,C 180,E1 13418.535,E2 13418.535} C_VEL
LIN {X 0,Y 339.697,Z 958.842,A -85,B 0,C 180,E1 13425.511,E2 13425.511} C_VEL
LIN {X 0,Y 345.091,Z 944.403,A -85,B 0,C 180,E1 13431.896,E2 13431.896} C_VEL
LIN {X 0,Y 353.066,Z 924.164,A -85,B 0,C 180,E1 13437.797,E2 13437.797} C_VEL
LIN {X 0,Y 361.863,Z 900.37,A -85,B 0,C 180,E1 13442.594,E2 13442.594} C_VEL
LIN {X 0,Y 371.11,Z 872.164,A -85,B 0,C 180,E1 13446.63,E2 13446.63} C_VEL
LIN {X 0,Y 379.729,Z 840.494,A -85,B 0,C 180,E1 13449.819,E2 13449.819} C_VEL
LIN {X 0,Y 380.601,Z 834.588,A -85,B 0,C 180,E1 13450.395,E2 13450.395} C_VEL
LIN {X 0,Y 371.257,Z 805.865,A -85,B 0,C 180,E1 13455.011,E2 13455.011} C_VEL
LIN {X 0,Y 358.582,Z 778.909,A -85,B 0,C 180,E1 13459.779,E2 13459.779} C_VEL
LIN {X 0,Y 344.851,Z 757.179,A -85,B 0,C 180,E1 13464.52,E2 13464.52} C_VEL
LIN {X 0,Y 339.314,Z 749.842,A -85,B 0,C 180,E1 13466.496,E2 13466.496} C_VEL
LIN {X 0,Y 335.539,Z 744.199,A -85,B 0,C 180,E1 13467.942,E2 13467.942} C_VEL
LIN {X 0,Y 331.956,Z 739.414,A -85,B 0,C 180,E1 13469.39,E2 13469.39} C_VEL
LIN {X 0,Y 331.722,Z 737.44,A -85,B 0,C 180,E1 13469.706,E2 13469.706} C_VEL
LIN {X 0,Y 331.953,Z 737.44,A -85,B 0,C 180,E1 13475.808,E2 13475.808} C_VEL
LIN {X 0,Y 332.526,Z 737.44,A -85,B 0,C 180,E1 13484.155,E2 13484.155} C_VEL
LIN {X 0,Y 332.959,Z 737.44,A -85,B 0,C 180,E1 13492.167,E2 13492.167} C_VEL
LIN {X 0,Y 333.432,Z 737.44,A -85,B 0,C 180,E1 13500.007,E2 13500.007} C_VEL
LIN {X 0,Y 332.911,Z 737.44,A -85,B 0,C 180,E1 13507.848,E2 13507.848} C_VEL
LIN {X 0,Y 332.379,Z 737.44,A -85,B 0,C 180,E1 13515.866,E2 13515.866} C_VEL
LIN {X 0,Y 332.207,Z 737.48,A -85,B 0,C 180,E1 13520.639,E2 13520.639} C_VEL
LIN {X 0,Y 334.011,Z 742.581,A -85,B 0,C 180,E1 13521.528,E2 13521.528} C_VEL
LIN {X 0,Y 337.299,Z 745.983,A -85,B 0,C 180,E1 13522.782,E2 13522.782} C_VEL
LIN {X 0,Y 351.82,Z 767.272,A -85,B 0,C 180,E1 13527.821,E2 13527.821} C_VEL
LIN {X 0,Y 368.309,Z 793.96,A -85,B 0,C 180,E1 13532.568,E2 13532.568} C_VEL
LIN {X 0,Y 382.198,Z 823.412,A -85,B 0,C 180,E1 13536.547,E2 13536.547} C_VEL
LIN {X 0,Y 387.211,Z 841.618,A -85,B 0,C 180,E1 13538.433,E2 13538.433} C_VEL
LIN {X 0,Y 379.225,Z 885.362,A -85,B 0,C 180,E1 13540.768,E2 13540.768} C_VEL
LIN {X 0,Y 369.569,Z 927.267,A -85,B 0,C 180,E1 13544.145,E2 13544.145} C_VEL
LIN {X 0,Y 359.878,Z 964.401,A -85,B 0,C 180,E1 13548.342,E2 13548.342} C_VEL
LIN {X 0,Y 350.757,Z 998.586,A -85,B 0,C 180,E1 13553.594,E2 13553.594} C_VEL
LIN {X 0,Y 343.355,Z 1027.977,A -85,B 0,C 180,E1 13559.639,E2 13559.639} C_VEL
LIN {X 0,Y 338.3,Z 1051.909,A -85,B 0,C 180,E1 13566.248,E2 13566.248} C_VEL
LIN {X 0,Y 335.658,Z 1069.517,A -85,B 0,C 180,E1 13572.951,E2 13572.951} C_VEL
LIN {X 0,Y 334.563,Z 1081.065,A -85,B 0,C 180,E1 13579.571,E2 13579.571} C_VEL
LIN {X 0,Y 334.438,Z 1086.368,A -85,B 0,C 180,E1 13584.854,E2 13584.854} C_VEL
LIN {X 0,Y 334.574,Z 1088.114,A -85,B 0,C 180,E1 13590,E2 13590} C_VEL
LIN {X 0,Y 334.389,Z 1085.285,A -85,B 0,C 180,E1 13596.499,E2 13596.499} C_VEL
LIN {X 0,Y 334.859,Z 1077.112,A -85,B 0,C 180,E1 13603.065,E2 13603.065} C_VEL
LIN {X 0,Y 336.285,Z 1064.339,A -85,B 0,C 180,E1 13609.275,E2 13609.275} C_VEL
LIN {X 0,Y 337.924,Z 1053.959,A -85,B 0,C 180,E1 13613.073,E2 13613.073} C_VEL
LIN {X 0,Y 335.415,Z 1045.901,A -85,B 0,C 180,E1 13615.694,E2 13615.694} C_VEL
LIN {X 0,Y 333.487,Z 1037.203,A -85,B 0,C 180,E1 13618.291,E2 13618.291} C_VEL
LIN {X 0,Y 340.088,Z 1010.957,A -85,B 0,C 180,E1 13624.537,E2 13624.537} C_VEL
LIN {X 0,Y 348.985,Z 979.215,A -85,B 0,C 180,E1 13630.189,E2 13630.189} C_VEL
LIN {X 0,Y 358.73,Z 944.426,A -85,B 0,C 180,E1 13634.799,E2 13634.799} C_VEL
LIN {X 0,Y 368.402,Z 907.055,A -85,B 0,C 180,E1 13638.427,E2 13638.427} C_VEL
LIN {X 0,Y 377.148,Z 867.205,A -85,B 0,C 180,E1 13641.163,E2 13641.163} C_VEL
LIN {X 0,Y 381.271,Z 842.028,A -85,B 0,C 180,E1 13642.471,E2 13642.471} C_VEL
LIN {X 0,Y 373.857,Z 819.867,A -85,B 0,C 180,E1 13645.102,E2 13645.102} C_VEL
LIN {X 0,Y 359.847,Z 791.674,A -85,B 0,C 180,E1 13649.331,E2 13649.331} C_VEL
LIN {X 0,Y 343.008,Z 764.736,A -85,B 0,C 180,E1 13654.68,E2 13654.68} C_VEL
LIN {X 0,Y 332.769,Z 750.68,A -85,B 0,C 180,E1 13658.547,E2 13658.547} C_VEL
LIN {X 0,Y 328.481,Z 744.386,A -85,B 0,C 180,E1 13660.429,E2 13660.429} C_VEL
LIN {X 0,Y 324.697,Z 739.794,A -85,B 0,C 180,E1 13662.206,E2 13662.206} C_VEL
LIN {X 0,Y 324.35,Z 737.44,A -85,B 0,C 180,E1 13662.678,E2 13662.678} C_VEL
LIN {X 0,Y 324.686,Z 737.44,A -85,B 0,C 180,E1 13669.244,E2 13669.244} C_VEL
LIN {X 0,Y 325.415,Z 737.44,A -85,B 0,C 180,E1 13677.327,E2 13677.327} C_VEL
LIN {X 0,Y 325.348,Z 737.44,A -85,B 0,C 180,E1 13682.66,E2 13682.66} C_VEL
LIN {X 0,Y 324.75,Z 737.44,A -85,B 0,C 180,E1 13690.739,E2 13690.739} C_VEL
LIN {X 0,Y 324.3,Z 737.44,A -85,B 0,C 180,E1 13699.065,E2 13699.065} C_VEL
LIN {X 0,Y 323.988,Z 738.142,A -85,B 0,C 180,E1 13707.265,E2 13707.265} C_VEL
LIN {X 0,Y 326.276,Z 743.13,A -85,B 0,C 180,E1 13708.475,E2 13708.475} C_VEL
LIN {X 0,Y 329.408,Z 746.165,A -85,B 0,C 180,E1 13709.833,E2 13709.833} C_VEL
LIN {X 0,Y 340.777,Z 762.288,A -85,B 0,C 180,E1 13714.395,E2 13714.395} C_VEL
LIN {X 0,Y 353.814,Z 783.415,A -85,B 0,C 180,E1 13719.267,E2 13719.267} C_VEL
LIN {X 0,Y 365.342,Z 808.463,A -85,B 0,C 180,E1 13723.948,E2 13723.948} C_VEL
LIN {X 0,Y 374.106,Z 836.331,A -85,B 0,C 180,E1 13728.594,E2 13728.594} C_VEL
LIN {X 0,Y 374.183,Z 841.295,A -85,B 0,C 180,E1 13729.239,E2 13729.239} C_VEL
LIN {X 0,Y 365.521,Z 872.11,A -85,B 0,C 180,E1 13732.342,E2 13732.342} C_VEL
LIN {X 0,Y 355.915,Z 900.613,A -85,B 0,C 180,E1 13736.428,E2 13736.428} C_VEL
LIN {X 0,Y 346.074,Z 925.974,A -85,B 0,C 180,E1 13741.592,E2 13741.592} C_VEL
LIN {X 0,Y 337.757,Z 946.061,A -85,B 0,C 180,E1 13747.604,E2 13747.604} C_VEL
LIN {X 0,Y 332.1,Z 960.402,A -85,B 0,C 180,E1 13754.126,E2 13754.126} C_VEL
LIN {X 0,Y 329.1,Z 969.108,A -85,B 0,C 180,E1 13760.734,E2 13760.734} C_VEL
LIN {X 0,Y 328.126,Z 972.982,A -85,B 0,C 180,E1 13767.356,E2 13767.356} C_VEL
LIN {X 0,Y 328.13,Z 972.947,A -85,B 0,C 180,E1 13772.645,E2 13772.645} C_VEL
LIN {X 0,Y 329.019,Z 969.524,A -85,B 0,C 180,E1 13778.737,E2 13778.737} C_VEL
LIN {X 0,Y 332.164,Z 960.217,A -85,B 0,C 180,E1 13785.871,E2 13785.871} C_VEL
LIN {X 0,Y 337.843,Z 945.8,A -85,B 0,C 180,E1 13792.391,E2 13792.391} C_VEL
LIN {X 0,Y 345.674,Z 926.819,A -85,B 0,C 180,E1 13798.088,E2 13798.088} C_VEL
LIN {X 0,Y 355.35,Z 901.89,A -85,B 0,C 180,E1 13803.268,E2 13803.268} C_VEL
LIN {X 0,Y 364.942,Z 873.802,A -85,B 0,C 180,E1 13807.354,E2 13807.354} C_VEL
LIN {X 0,Y 373.971,Z 841.893,A -85,B 0,C 180,E1 13810.611,E2 13810.611} C_VEL
LIN {X 0,Y 374.371,Z 837.343,A -85,B 0,C 180,E1 13811.121,E2 13811.121} C_VEL
LIN {X 0,Y 365.882,Z 810.065,A -85,B 0,C 180,E1 13815.668,E2 13815.668} C_VEL
LIN {X 0,Y 353.799,Z 783.361,A -85,B 0,C 180,E1 13820.613,E2 13820.613} C_VEL
LIN {X 0,Y 340.873,Z 762.502,A -85,B 0,C 180,E1 13825.423,E2 13825.423} C_VEL
LIN {X 0,Y 332.434,Z 750.692,A -85,B 0,C 180,E1 13828.714,E2 13828.714} C_VEL
LIN {X 0,Y 327.926,Z 744.336,A -85,B 0,C 180,E1 13830.658,E2 13830.658} C_VEL
LIN {X 0,Y 324.313,Z 740.018,A -85,B 0,C 180,E1 13832.329,E2 13832.329} C_VEL
LIN {X 0,Y 323.955,Z 737.44,A -85,B 0,C 180,E1 13832.737,E2 13832.737} C_VEL
LIN {X 0,Y 324.348,Z 737.44,A -85,B 0,C 180,E1 13840.938,E2 13840.938} C_VEL
LIN {X 0,Y 324.747,Z 737.44,A -85,B 0,C 180,E1 13848.247,E2 13848.247} C_VEL
LIN {X 0,Y 325.2,Z 737.44,A -85,B 0,C 180,E1 13854.665,E2 13854.665} C_VEL
LIN {X 0,Y 325.546,Z 737.44,A -85,B 0,C 180,E1 13860.007,E2 13860.007} C_VEL
LIN {X 0,Y 324.965,Z 737.44,A -85,B 0,C 180,E1 13868.041,E2 13868.041} C_VEL
LIN {X 0,Y 324.443,Z 737.44,A -85,B 0,C 180,E1 13876.265,E2 13876.265} C_VEL
LIN {X 0,Y 324.395,Z 738.232,A -85,B 0,C 180,E1 13877.65,E2 13877.65} C_VEL
LIN {X 0,Y 326.945,Z 743.323,A -85,B 0,C 180,E1 13878.977,E2 13878.977} C_VEL
LIN {X 0,Y 329.71,Z 746.034,A -85,B 0,C 180,E1 13880.179,E2 13880.179} C_VEL
LIN {X 0,Y 343.503,Z 765.703,A -85,B 0,C 180,E1 13885.543,E2 13885.543} C_VEL
LIN {X 0,Y 359.559,Z 791.325,A -85,B 0,C 180,E1 13890.619,E2 13890.619} C_VEL
LIN {X 0,Y 373.382,Z 818.728,A -85,B 0,C 180,E1 13894.765,E2 13894.765} C_VEL
LIN {X 0,Y 381.272,Z 842.108,A -85,B 0,C 180,E1 13897.549,E2 13897.549} C_VEL
LIN {X 0,Y 373.05,Z 886.736,A -85,B 0,C 180,E1 13900.047,E2 13900.047} C_VEL
LIN {X 0,Y 363.255,Z 927.201,A -85,B 0,C 180,E1 13903.378,E2 13903.378} C_VEL
LIN {X 0,Y 353.174,Z 964.028,A -85,B 0,C 180,E1 13907.619,E2 13907.619} C_VEL
LIN {X 0,Y 343.899,Z 997.323,A -85,B 0,C 180,E1 13912.834,E2 13912.834} C_VEL
LIN {X 0,Y 336.201,Z 1026.056,A -85,B 0,C 180,E1 13918.833,E2 13918.833} C_VEL
LIN {X 0,Y 330.706,Z 1050.378,A -85,B 0,C 180,E1 13925.668,E2 13925.668} C_VEL
LIN {X 0,Y 327.898,Z 1068.057,A -85,B 0,C 180,E1 13932.535,E2 13932.535} C_VEL
LIN {X 0,Y 326.758,Z 1079.661,A -85,B 0,C 180,E1 13939.319,E2 13939.319} C_VEL
LIN {X 0,Y 326.644,Z 1084.965,A -85,B 0,C 180,E1 13944.681,E2 13944.681} C_VEL
LIN {X 0,Y 326.793,Z 1086.766,A -85,B 0,C 180,E1 13950,E2 13950} C_VEL
LIN {X 0,Y 326.602,Z 1083.917,A -85,B 0,C 180,E1 13956.655,E2 13956.655} C_VEL
LIN {X 0,Y 327.063,Z 1075.686,A -85,B 0,C 180,E1 13963.382,E2 13963.382} C_VEL
LIN {X 0,Y 328.667,Z 1061.761,A -85,B 0,C 180,E1 13970.211,E2 13970.211} C_VEL
LIN {X 0,Y 332.839,Z 1040.091,A -85,B 0,C 180,E1 13977.498,E2 13977.498} C_VEL
LIN {X 0,Y 333.487,Z 1037.203,A -85,B 0,C 180,E1 13978.291,E2 13978.291} C_VEL
LIN {X 0,Y 331.845,Z 1028.08,A -85,B 0,C 180,E1 13980.856,E2 13980.856} C_VEL
LIN {X 0,Y 330.625,Z 1018.36,A -85,B 0,C 180,E1 13983.379,E2 13983.379} C_VEL
LIN {X 0,Y 338.887,Z 989.62,A -85,B 0,C 180,E1 13989.123,E2 13989.123} C_VEL
LIN {X 0,Y 348.537,Z 956.996,A -85,B 0,C 180,E1 13994.028,E2 13994.028} C_VEL
LIN {X 0,Y 358.969,Z 920.095,A -85,B 0,C 180,E1 13998.103,E2 13998.103} C_VEL
LIN {X 0,Y 368.892,Z 879.902,A -85,B 0,C 180,E1 14001.241,E2 14001.241} C_VEL
LIN {X 0,Y 375.433,Z 844.677,A -85,B 0,C 180,E1 14003.222,E2 14003.222} C_VEL
LIN {X 0,Y 367.962,Z 822.244,A -85,B 0,C 180,E1 14006.043,E2 14006.043} C_VEL
LIN {X 0,Y 354.937,Z 795.67,A -85,B 0,C 180,E1 14010.268,E2 14010.268} C_VEL
LIN {X 0,Y 339.661,Z 770.906,A -85,B 0,C 180,E1 14015.382,E2 14015.382} C_VEL
LIN {X 0,Y 329.787,Z 757.155,A -85,B 0,C 180,E1 14019.269,E2 14019.269} C_VEL
LIN {X 0,Y 325.779,Z 751.334,A -85,B 0,C 180,E1 14021.096,E2 14021.096} C_VEL
LIN {X 0,Y 321.922,Z 745.333,A -85,B 0,C 180,E1 14023.066,E2 14023.066} C_VEL
LIN {X 0,Y 317.029,Z 740.198,A -85,B 0,C 180,E1 14025.739,E2 14025.739} C_VEL
LIN {X 0,Y 316.619,Z 737.44,A -85,B 0,C 180,E1 14026.4,E2 14026.4} C_VEL
LIN {X 0,Y 317.219,Z 737.44,A -85,B 0,C 180,E1 14034.516,E2 14034.516} C_VEL
LIN {X 0,Y 317.658,Z 737.44,A -85,B 0,C 180,E1 14039.993,E2 14039.993} C_VEL
LIN {X 0,Y 317.02,Z 737.44,A -85,B 0,C 180,E1 14048.229,E2 14048.229} C_VEL
LIN {X 0,Y 316.491,Z 737.44,A -85,B 0,C 180,E1 14056.671,E2 14056.671} C_VEL
LIN {X 0,Y 316.094,Z 738.176,A -85,B 0,C 180,E1 14063.485,E2 14063.485} C_VEL
LIN {X 0,Y 318.367,Z 742.998,A -85,B 0,C 180,E1 14064.962,E2 14064.962} C_VEL
LIN {X 0,Y 321.75,Z 745.9,A -85,B 0,C 180,E1 14066.707,E2 14066.707} C_VEL
LIN {X 0,Y 325.819,Z 751.651,A -85,B 0,C 180,E1 14068.717,E2 14068.717} C_VEL
LIN {X 0,Y 336.981,Z 767.699,A -85,B 0,C 180,E1 14073.574,E2 14073.574} C_VEL
LIN {X 0,Y 349.705,Z 789.249,A -85,B 0,C 180,E1 14078.721,E2 14078.721} C_VEL
LIN {X 0,Y 360.859,Z 814.887,A -85,B 0,C 180,E1 14083.662,E2 14083.662} C_VEL
LIN {X 0,Y 368.568,Z 841.861,A -85,B 0,C 180,E1 14088.324,E2 14088.324} C_VEL
LIN {X 0,Y 359.422,Z 873.818,A -85,B 0,C 180,E1 14091.603,E2 14091.603} C_VEL
LIN {X 0,Y 349.485,Z 902.118,A -85,B 0,C 180,E1 14095.725,E2 14095.725} C_VEL
LIN {X 0,Y 339.216,Z 927.398,A -85,B 0,C 180,E1 14100.963,E2 14100.963} C_VEL
LIN {X 0,Y 331.092,Z 946.174,A -85,B 0,C 180,E1 14106.603,E2 14106.603} C_VEL
LIN {X 0,Y 325.14,Z 960.385,A -85,B 0,C 180,E1 14112.948,E2 14112.948} C_VEL
LIN {X 0,Y 321.9,Z 969.128,A -85,B 0,C 180,E1 14119.156,E2 14119.156} C_VEL
LIN {X 0,Y 320.48,Z 973.317,A -85,B 0,C 180,E1 14124.579,E2 14124.579} C_VEL
LIN {X 0,Y 320.447,Z 974.657,A -85,B 0,C 180,E1 14130,E2 14130} C_VEL
LIN {X 0,Y 320.503,Z 973.258,A -85,B 0,C 180,E1 14135.421,E2 14135.421} C_VEL
LIN {X 0,Y 322.461,Z 967.448,A -85,B 0,C 180,E1 14142.198,E2 14142.198} C_VEL
LIN {X 0,Y 326.684,Z 956.57,A -85,B 0,C 180,E1 14148.93,E2 14148.93} C_VEL
LIN {X 0,Y 333.939,Z 939.628,A -85,B 0,C 180,E1 14155.511,E2 14155.511} C_VEL
LIN {X 0,Y 342.936,Z 918.366,A -85,B 0,C 180,E1 14161.036,E2 14161.036} C_VEL
LIN {X 0,Y 352.709,Z 893.133,A -85,B 0,C 180,E1 14165.65,E2 14165.65} C_VEL
LIN {X 0,Y 362.329,Z 864.551,A -85,B 0,C 180,E1 14169.357,E2 14169.357} C_VEL
LIN {X 0,Y 368.449,Z 841.322,A -85,B 0,C 180,E1 14171.655,E2 14171.655} C_VEL
LIN {X 0,Y 360.379,Z 813.835,A -85,B 0,C 180,E1 14176.424,E2 14176.424} C_VEL
LIN {X 0,Y 348.916,Z 787.8,A -85,B 0,C 180,E1 14181.472,E2 14181.472} C_VEL
LIN {X 0,Y 335.453,Z 765.113,A -85,B 0,C 180,E1 14186.939,E2 14186.939} C_VEL
LIN {X 0,Y 325.327,Z 751.3,A -85,B 0,C 180,E1 14191.33,E2 14191.33} C_VEL
LIN {X 0,Y 321.638,Z 745.657,A -85,B 0,C 180,E1 14193.18,E2 14193.18} C_VEL
LIN {X 0,Y 316.43,Z 739.897,A -85,B 0,C 180,E1 14196.029,E2 14196.029} C_VEL
LIN {X 0,Y 316.057,Z 737.44,A -85,B 0,C 180,E1 14196.569,E2 14196.569} C_VEL
LIN {X 0,Y 316.589,Z 737.44,A -85,B 0,C 180,E1 14203.335,E2 14203.335} C_VEL
LIN {X 0,Y 317.079,Z 737.44,A -85,B 0,C 180,E1 14211.772,E2 14211.772} C_VEL
LIN {X 0,Y 317.664,Z 737.44,A -85,B 0,C 180,E1 14220.007,E2 14220.007} C_VEL
LIN {X 0,Y 317.018,Z 737.44,A -85,B 0,C 180,E1 14228.244,E2 14228.244} C_VEL
LIN {X 0,Y 316.638,Z 738.163,A -85,B 0,C 180,E1 14234.014,E2 14234.014} C_VEL
LIN {X 0,Y 318.923,Z 743.13,A -85,B 0,C 180,E1 14235.494,E2 14235.494} C_VEL
LIN {X 0,Y 322.065,Z 745.834,A -85,B 0,C 180,E1 14237.107,E2 14237.107} C_VEL
LIN {X 0,Y 326.291,Z 751.718,A -85,B 0,C 180,E1 14239.189,E2 14239.189} C_VEL
LIN {X 0,Y 340.561,Z 772.24,A -85,B 0,C 180,E1 14244.987,E2 14244.987} C_VEL
LIN {X 0,Y 356.55,Z 798.584,A -85,B 0,C 180,E1 14250.285,E2 14250.285} C_VEL
LIN {X 0,Y 369.458,Z 825.932,A -85,B 0,C 180,E1 14254.477,E2 14254.477} C_VEL
LIN {X 0,Y 375.556,Z 845.331,A -85,B 0,C 180,E1 14256.864,E2 14256.864} C_VEL
LIN {X 0,Y 367.019,Z 887.636,A -85,B 0,C 180,E1 14259.27,E2 14259.27} C_VEL
LIN {X 0,Y 357.177,Z 926.455,A -85,B 0,C 180,E1 14262.511,E2 14262.511} C_VEL
LIN {X 0,Y 346.767,Z 962.954,A -85,B 0,C 180,E1 14266.771,E2 14266.771} C_VEL
LIN {X 0,Y 336.988,Z 996.29,A -85,B 0,C 180,E1 14272.08,E2 14272.08} C_VEL
LIN {X 0,Y 328.972,Z 1024.463,A -85,B 0,C 180,E1 14278.068,E2 14278.068} C_VEL
LIN {X 0,Y 323.151,Z 1048.859,A -85,B 0,C 180,E1 14285.061,E2 14285.061} C_VEL
LIN {X 0,Y 320.107,Z 1066.81,A -85,B 0,C 180,E1 14292.203,E2 14292.203} C_VEL
LIN {X 0,Y 318.945,Z 1078.26,A -85,B 0,C 180,E1 14299.054,E2 14299.054} C_VEL
LIN {X 0,Y 318.848,Z 1083.601,A -85,B 0,C 180,E1 14304.55,E2 14304.55} C_VEL
LIN {X 0,Y 319.03,Z 1085.422,A -85,B 0,C 180,E1 14310,E2 14310} C_VEL
LIN {X 0,Y 318.799,Z 1082.548,A -85,B 0,C 180,E1 14316.818,E2 14316.818} C_VEL
LIN {X 0,Y 319.281,Z 1074.267,A -85,B 0,C 180,E1 14323.715,E2 14323.715} C_VEL
LIN {X 0,Y 320.954,Z 1060.27,A -85,B 0,C 180,E1 14330.719,E2 14330.719} C_VEL
LIN {X 0,Y 325.35,Z 1038.782,A -85,B 0,C 180,E1 14338.109,E2 14338.109} C_VEL
LIN {X 0,Y 330.625,Z 1018.36,A -85,B 0,C 180,E1 14343.379,E2 14343.379} C_VEL
LIN {X 0,Y 329.871,Z 1008.226,A -85,B 0,C 180,E1 14345.857,E2 14345.857} C_VEL
LIN {X 0,Y 329.455,Z 997.54,A -85,B 0,C 180,E1 14348.276,E2 14348.276} C_VEL
LIN {X 0,Y 339.565,Z 964.823,A -85,B 0,C 180,E1 14353.7,E2 14353.7} C_VEL
LIN {X 0,Y 350.304,Z 929.315,A -85,B 0,C 180,E1 14358.011,E2 14358.011} C_VEL
LIN {X 0,Y 360.345,Z 892.156,A -85,B 0,C 180,E1 14361.262,E2 14361.262} C_VEL
LIN {X 0,Y 368.881,Z 853.52,A -85,B 0,C 180,E1 14363.624,E2 14363.624} C_VEL
LIN {X 0,Y 369.743,Z 847.918,A -85,B 0,C 180,E1 14363.919,E2 14363.919} C_VEL
LIN {X 0,Y 362.663,Z 825.94,A -85,B 0,C 180,E1 14366.834,E2 14366.834} C_VEL
LIN {X 0,Y 349.703,Z 798.888,A -85,B 0,C 180,E1 14371.324,E2 14371.324} C_VEL
LIN {X 0,Y 335.682,Z 776.054,A -85,B 0,C 180,E1 14376.358,E2 14376.358} C_VEL
LIN {X 0,Y 323.758,Z 758.653,A -85,B 0,C 180,E1 14381.493,E2 14381.493} C_VEL
LIN {X 0,Y 318.359,Z 751.562,A -85,B 0,C 180,E1 14384.301,E2 14384.301} C_VEL
LIN {X 0,Y 314.613,Z 746.033,A -85,B 0,C 180,E1 14386.603,E2 14386.603} C_VEL
LIN {X 0,Y 309.231,Z 739.671,A -85,B 0,C 180,E1 14390.482,E2 14390.482} C_VEL
LIN {X 0,Y 308.994,Z 737.44,A -85,B 0,C 180,E1 14391.186,E2 14391.186} C_VEL
LIN {X 0,Y 309.583,Z 737.44,A -85,B 0,C 180,E1 14397.19,E2 14397.19} C_VEL
LIN {X 0,Y 309.541,Z 737.44,A -85,B 0,C 180,E1 14402.796,E2 14402.796} C_VEL
LIN {X 0,Y 308.857,Z 737.44,A -85,B 0,C 180,E1 14411.369,E2 14411.369} C_VEL
LIN {X 0,Y 308.472,Z 738.144,A -85,B 0,C 180,E1 14418.687,E2 14418.687} C_VEL
LIN {X 0,Y 310.98,Z 743.408,A -85,B 0,C 180,E1 14420.865,E2 14420.865} C_VEL
LIN {X 0,Y 314.167,Z 745.908,A -85,B 0,C 180,E1 14422.948,E2 14422.948} C_VEL
LIN {X 0,Y 318.102,Z 751.663,A -85,B 0,C 180,E1 14425.353,E2 14425.353} C_VEL
LIN {X 0,Y 320.197,Z 754.339,A -85,B 0,C 180,E1 14426.483,E2 14426.483} C_VEL
LIN {X 0,Y 329.454,Z 767.332,A -85,B 0,C 180,E1 14431.024,E2 14431.024} C_VEL
LIN {X 0,Y 341.141,Z 786.692,A -85,B 0,C 180,E1 14436.204,E2 14436.204} C_VEL
LIN {X 0,Y 352.268,Z 810.142,A -85,B 0,C 180,E1 14441.279,E2 14441.279} C_VEL
LIN {X 0,Y 360.957,Z 837.987,A -85,B 0,C 180,E1 14446.378,E2 14446.378} C_VEL
LIN {X 0,Y 362.204,Z 846.861,A -85,B 0,C 180,E1 14447.822,E2 14447.822} C_VEL
LIN {X 0,Y 352.268,Z 878.893,A -85,B 0,C 180,E1 14451.254,E2 14451.254} C_VEL
LIN {X 0,Y 341.726,Z 907.019,A -85,B 0,C 180,E1 14455.606,E2 14455.606} C_VEL
LIN {X 0,Y 331.872,Z 930.023,A -85,B 0,C 180,E1 14460.633,E2 14460.633} C_VEL
LIN {X 0,Y 323.172,Z 949.293,A -85,B 0,C 180,E1 14466.727,E2 14466.727} C_VEL
LIN {X 0,Y 317.082,Z 963.143,A -85,B 0,C 180,E1 14473.353,E2 14473.353} C_VEL
LIN {X 0,Y 313.717,Z 971.819,A -85,B 0,C 180,E1 14480.276,E2 14480.276} C_VEL
LIN {X 0,Y 312.578,Z 975.678,A -85,B 0,C 180,E1 14487.224,E2 14487.224} C_VEL
LIN {X 0,Y 312.583,Z 975.645,A -85,B 0,C 180,E1 14492.776,E2 14492.776} C_VEL
LIN {X 0,Y 313.77,Z 971.711,A -85,B 0,C 180,E1 14499.723,E2 14499.723} C_VEL
LIN {X 0,Y 317.142,Z 962.963,A -85,B 0,C 180,E1 14506.645,E2 14506.645} C_VEL
LIN {X 0,Y 323.33,Z 948.887,A -85,B 0,C 180,E1 14513.324,E2 14513.324} C_VEL
LIN {X 0,Y 331.997,Z 929.667,A -85,B 0,C 180,E1 14519.356,E2 14519.356} C_VEL
LIN {X 0,Y 342.486,Z 904.911,A -85,B 0,C 180,E1 14524.691,E2 14524.691} C_VEL
LIN {X 0,Y 353.184,Z 875.862,A -85,B 0,C 180,E1 14529.021,E2 14529.021} C_VEL
LIN {X 0,Y 362.342,Z 844.321,A -85,B 0,C 180,E1 14532.38,E2 14532.38} C_VEL
LIN {X 0,Y 354.83,Z 817.372,A -85,B 0,C 180,E1 14537.251,E2 14537.251} C_VEL
LIN {X 0,Y 344.115,Z 792.406,A -85,B 0,C 180,E1 14542.326,E2 14542.326} C_VEL
LIN {X 0,Y 332.079,Z 771.419,A -85,B 0,C 180,E1 14547.62,E2 14547.62} C_VEL
LIN {X 0,Y 322.661,Z 758.058,A -85,B 0,C 180,E1 14552.027,E2 14552.027} C_VEL
LIN {X 0,Y 318.415,Z 751.854,A -85,B 0,C 180,E1 14554.301,E2 14554.301} C_VEL
LIN {X 0,Y 314.248,Z 746.274,A -85,B 0,C 180,E1 14556.777,E2 14556.777} C_VEL
LIN {X 0,Y 312.165,Z 744.251,A -85,B 0,C 180,E1 14558.129,E2 14558.129} C_VEL
LIN {X 0,Y 308.746,Z 739.488,A -85,B 0,C 180,E1 14560.773,E2 14560.773} C_VEL
LIN {X 0,Y 308.475,Z 737.44,A -85,B 0,C 180,E1 14561.406,E2 14561.406} C_VEL
LIN {X 0,Y 308.963,Z 737.44,A -85,B 0,C 180,E1 14568.705,E2 14568.705} C_VEL
LIN {X 0,Y 309.544,Z 737.44,A -85,B 0,C 180,E1 14577.204,E2 14577.204} C_VEL
LIN {X 0,Y 309.586,Z 737.44,A -85,B 0,C 180,E1 14582.81,E2 14582.81} C_VEL
LIN {X 0,Y 308.984,Z 738.178,A -85,B 0,C 180,E1 14589.348,E2 14589.348} C_VEL
LIN {X 0,Y 311.262,Z 743.088,A -85,B 0,C 180,E1 14591.314,E2 14591.314} C_VEL
LIN {X 0,Y 314.596,Z 745.926,A -85,B 0,C 180,E1 14593.486,E2 14593.486} C_VEL
LIN {X 0,Y 318.219,Z 751.458,A -85,B 0,C 180,E1 14595.706,E2 14595.706} C_VEL
LIN {X 0,Y 320.457,Z 754.378,A -85,B 0,C 180,E1 14596.924,E2 14596.924} C_VEL
LIN {X 0,Y 326.659,Z 763.215,A -85,B 0,C 180,E1 14599.964,E2 14599.964} C_VEL
LIN {X 0,Y 337.67,Z 778.865,A -85,B 0,C 180,E1 14604.431,E2 14604.431} C_VEL
LIN {X 0,Y 352.538,Z 804.322,A -85,B 0,C 180,E1 14609.694,E2 14609.694} C_VEL
LIN {X 0,Y 364.736,Z 831.391,A -85,B 0,C 180,E1 14613.977,E2 14613.977} C_VEL
LIN {X 0,Y 369.608,Z 848.689,A -85,B 0,C 180,E1 14616.137,E2 14616.137} C_VEL
LIN {X 0,Y 360.952,Z 889.021,A -85,B 0,C 180,E1 14618.504,E2 14618.504} C_VEL
LIN {X 0,Y 350.663,Z 927.665,A -85,B 0,C 180,E1 14621.819,E2 14621.819} C_VEL
LIN {X 0,Y 339.917,Z 963.518,A -85,B 0,C 180,E1 14626.119,E2 14626.119} C_VEL
LIN {X 0,Y 330.073,Z 995.539,A -85,B 0,C 180,E1 14631.348,E2 14631.348} C_VEL
LIN {X 0,Y 321.391,Z 1024.366,A -85,B 0,C 180,E1 14637.654,E2 14637.654} C_VEL
LIN {X 0,Y 315.574,Z 1047.337,A -85,B 0,C 180,E1 14644.419,E2 14644.419} C_VEL
LIN {X 0,Y 312.345,Z 1065.53,A -85,B 0,C 180,E1 14651.834,E2 14651.834} C_VEL
LIN {X 0,Y 311.146,Z 1076.863,A -85,B 0,C 180,E1 14658.776,E2 14658.776} C_VEL
LIN {X 0,Y 311.056,Z 1082.239,A -85,B 0,C 180,E1 14664.413,E2 14664.413} C_VEL
LIN {X 0,Y 311.246,Z 1084.074,A -85,B 0,C 180,E1 14670,E2 14670} C_VEL
LIN {X 0,Y 310.997,Z 1081.18,A -85,B 0,C 180,E1 14676.99,E2 14676.99} C_VEL
LIN {X 0,Y 311.457,Z 1072.843,A -85,B 0,C 180,E1 14684.066,E2 14684.066} C_VEL
LIN {X 0,Y 313.264,Z 1058.786,A -85,B 0,C 180,E1 14691.252,E2 14691.252} C_VEL
LIN {X 0,Y 317.985,Z 1037.234,A -85,B 0,C 180,E1 14698.821,E2 14698.821} C_VEL
LIN {X 0,Y 325.501,Z 1010.236,A -85,B 0,C 180,E1 14705.69,E2 14705.69} C_VEL
LIN {X 0,Y 329.455,Z 997.54,A -85,B 0,C 180,E1 14708.276,E2 14708.276} C_VEL
LIN {X 0,Y 329.43,Z 986.452,A -85,B 0,C 180,E1 14710.639,E2 14710.639} C_VEL
LIN {X 0,Y 329.762,Z 974.843,A -85,B 0,C 180,E1 14712.921,E2 14712.921} C_VEL
LIN {X 0,Y 340.383,Z 941.883,A -85,B 0,C 180,E1 14717.449,E2 14717.449} C_VEL
LIN {X 0,Y 351.165,Z 905.24,A -85,B 0,C 180,E1 14721.123,E2 14721.123} C_VEL
LIN {X 0,Y 361.104,Z 864.794,A -85,B 0,C 180,E1 14723.952,E2 14723.952} C_VEL
LIN {X 0,Y 363.77,Z 849.709,A -85,B 0,C 180,E1 14724.817,E2 14724.817} C_VEL
LIN {X 0,Y 356.146,Z 826.695,A -85,B 0,C 180,E1 14728.091,E2 14728.091} C_VEL
LIN {X 0,Y 343.231,Z 799.972,A -85,B 0,C 180,E1 14732.893,E2 14732.893} C_VEL
LIN {X 0,Y 329.916,Z 778.029,A -85,B 0,C 180,E1 14738.148,E2 14738.148} C_VEL
LIN {X 0,Y 320.606,Z 764.823,A -85,B 0,C 180,E1 14742.452,E2 14742.452} C_VEL
LIN {X 0,Y 316.306,Z 758.782,A -85,B 0,C 180,E1 14744.819,E2 14744.819} C_VEL
LIN {X 0,Y 311.376,Z 751.97,A -85,B 0,C 180,E1 14748.001,E2 14748.001} C_VEL
LIN {X 0,Y 307.485,Z 746.672,A -85,B 0,C 180,E1 14751.083,E2 14751.083} C_VEL
LIN {X 0,Y 306.313,Z 744.854,A -85,B 0,C 180,E1 14752.182,E2 14752.182} C_VEL
LIN {X 0,Y 302.075,Z 739.916,A -85,B 0,C 180,E1 14757.3,E2 14757.3} C_VEL
LIN {X 0,Y 301.698,Z 737.44,A -85,B 0,C 180,E1 14758.555,E2 14758.555} C_VEL
LIN {X 0,Y 301.397,Z 737.44,A -85,B 0,C 180,E1 14765.758,E2 14765.758} C_VEL
LIN {X 0,Y 301.008,Z 738.095,A -85,B 0,C 180,E1 14770.347,E2 14770.347} C_VEL
LIN {X 0,Y 303.423,Z 743.411,A -85,B 0,C 180,E1 14774.701,E2 14774.701} C_VEL
LIN {X 0,Y 306.918,Z 746.07,A -85,B 0,C 180,E1 14778.227,E2 14778.227} C_VEL
LIN {X 0,Y 310.545,Z 751.77,A -85,B 0,C 180,E1 14781.235,E2 14781.235} C_VEL
LIN {X 0,Y 312.572,Z 753.877,A -85,B 0,C 180,E1 14782.601,E2 14782.601} C_VEL
LIN {X 0,Y 318.368,Z 762.154,A -85,B 0,C 180,E1 14786.181,E2 14786.181} C_VEL
LIN {X 0,Y 326.865,Z 774.535,A -85,B 0,C 180,E1 14790.62,E2 14790.62} C_VEL
LIN {X 0,Y 337.486,Z 793.174,A -85,B 0,C 180,E1 14795.756,E2 14795.756} C_VEL
LIN {X 0,Y 347.577,Z 815.714,A -85,B 0,C 180,E1 14800.784,E2 14800.784} C_VEL
LIN {X 0,Y 354.982,Z 841.064,A -85,B 0,C 180,E1 14805.603,E2 14805.603} C_VEL
LIN {X 0,Y 356.55,Z 848.503,A -85,B 0,C 180,E1 14806.97,E2 14806.97} C_VEL
LIN {X 0,Y 346.005,Z 881.156,A -85,B 0,C 180,E1 14810.547,E2 14810.547} C_VEL
LIN {X 0,Y 335.336,Z 908.489,A -85,B 0,C 180,E1 14814.856,E2 14814.856} C_VEL
LIN {X 0,Y 325.089,Z 931.441,A -85,B 0,C 180,E1 14819.958,E2 14819.958} C_VEL
LIN {X 0,Y 316.038,Z 950.618,A -85,B 0,C 180,E1 14826.143,E2 14826.143} C_VEL
LIN {X 0,Y 309.591,Z 964.512,A -85,B 0,C 180,E1 14832.938,E2 14832.938} C_VEL
LIN {X 0,Y 306.037,Z 973.174,A -85,B 0,C 180,E1 14840.029,E2 14840.029} C_VEL
LIN {X 0,Y 304.815,Z 977.025,A -85,B 0,C 180,E1 14847.153,E2 14847.153} C_VEL
LIN {X 0,Y 304.821,Z 976.991,A -85,B 0,C 180,E1 14852.847,E2 14852.847} C_VEL
LIN {X 0,Y 306.097,Z 973.066,A -85,B 0,C 180,E1 14859.969,E2 14859.969} C_VEL
LIN {X 0,Y 309.651,Z 964.335,A -85,B 0,C 180,E1 14867.059,E2 14867.059} C_VEL
LIN {X 0,Y 316.197,Z 950.233,A -85,B 0,C 180,E1 14873.9,E2 14873.9} C_VEL
LIN {X 0,Y 325.229,Z 931.085,A -85,B 0,C 180,E1 14880.029,E2 14880.029} C_VEL
LIN {X 0,Y 336.143,Z 906.403,A -85,B 0,C 180,E1 14885.443,E2 14885.443} C_VEL
LIN {X 0,Y 347.217,Z 877.512,A -85,B 0,C 180,E1 14889.819,E2 14889.819} C_VEL
LIN {X 0,Y 356.344,Z 847.507,A -85,B 0,C 180,E1 14893.092,E2 14893.092} C_VEL
LIN {X 0,Y 349.204,Z 820.844,A -85,B 0,C 180,E1 14898.121,E2 14898.121} C_VEL
LIN {X 0,Y 339.303,Z 796.686,A -85,B 0,C 180,E1 14903.258,E2 14903.258} C_VEL
LIN {X 0,Y 328.415,Z 777.158,A -85,B 0,C 180,E1 14908.466,E2 14908.466} C_VEL
LIN {X 0,Y 320.326,Z 765.066,A -85,B 0,C 180,E1 14912.57,E2 14912.57} C_VEL
LIN {X 0,Y 315.971,Z 758.847,A -85,B 0,C 180,E1 14915.021,E2 14915.021} C_VEL
LIN {X 0,Y 311.313,Z 752.192,A -85,B 0,C 180,E1 14918.049,E2 14918.049} C_VEL
LIN {X 0,Y 307.292,Z 747.173,A -85,B 0,C 180,E1 14921.145,E2 14921.145} C_VEL
LIN {X 0,Y 306.422,Z 745.057,A -85,B 0,C 180,E1 14922.022,E2 14922.022} C_VEL
LIN {X 0,Y 301.445,Z 740.159,A -85,B 0,C 180,E1 14927.868,E2 14927.868} C_VEL
LIN {X 0,Y 301.061,Z 737.44,A -85,B 0,C 180,E1 14929.155,E2 14929.155} C_VEL
LIN {X 0,Y 301.649,Z 737.44,A -85,B 0,C 180,E1 14937.131,E2 14937.131} C_VEL
LIN {X 0,Y 301.71,Z 738.051,A -85,B 0,C 180,E1 14942.164,E2 14942.164} C_VEL
LIN {X 0,Y 303.868,Z 743.185,A -85,B 0,C 180,E1 14945.547,E2 14945.547} C_VEL
LIN {X 0,Y 307.289,Z 745.917,A -85,B 0,C 180,E1 14948.842,E2 14948.842} C_VEL
LIN {X 0,Y 310.768,Z 751.614,A -85,B 0,C 180,E1 14951.711,E2 14951.711} C_VEL
LIN {X 0,Y 312.865,Z 753.794,A -85,B 0,C 180,E1 14953.117,E2 14953.117} C_VEL
LIN {X 0,Y 318.755,Z 762.278,A -85,B 0,C 180,E1 14956.654,E2 14956.654} C_VEL
LIN {X 0,Y 327.326,Z 774.209,A -85,B 0,C 180,E1 14960.798,E2 14960.798} C_VEL
LIN {X 0,Y 340.963,Z 795.835,A -85,B 0,C 180,E1 14966.278,E2 14966.278} C_VEL
LIN {X 0,Y 354.685,Z 823.272,A -85,B 0,C 180,E1 14971.382,E2 14971.382} C_VEL
LIN {X 0,Y 363.35,Z 847.876,A -85,B 0,C 180,E1 14974.977,E2 14974.977} C_VEL
LIN {X 0,Y 363.473,Z 853.258,A -85,B 0,C 180,E1 14975.438,E2 14975.438} C_VEL
LIN {X 0,Y 353.718,Z 895.596,A -85,B 0,C 180,E1 14978.099,E2 14978.099} C_VEL
LIN {X 0,Y 342.177,Z 935.655,A -85,B 0,C 180,E1 14981.826,E2 14981.826} C_VEL
LIN {X 0,Y 330.605,Z 971.925,A -85,B 0,C 180,E1 14986.613,E2 14986.613} C_VEL
LIN {X 0,Y 320.181,Z 1003.81,A -85,B 0,C 180,E1 14992.389,E2 14992.389} C_VEL
LIN {X 0,Y 312.014,Z 1030.67,A -85,B 0,C 180,E1 14998.965,E2 14998.965} C_VEL
LIN {X 0,Y 306.677,Z 1052.214,A -85,B 0,C 180,E1 15006.108,E2 15006.108} C_VEL
LIN {X 0,Y 304.057,Z 1067.829,A -85,B 0,C 180,E1 15013.363,E2 15013.363} C_VEL
LIN {X 0,Y 303.239,Z 1077.13,A -85,B 0,C 180,E1 15019.936,E2 15019.936} C_VEL
LIN {X 0,Y 303.25,Z 1080.875,A -85,B 0,C 180,E1 15024.269,E2 15024.269} C_VEL
LIN {X 0,Y 303.483,Z 1082.729,A -85,B 0,C 180,E1 15030,E2 15030} C_VEL
LIN {X 0,Y 303.192,Z 1079.813,A -85,B 0,C 180,E1 15037.171,E2 15037.171} C_VEL
LIN {X 0,Y 303.565,Z 1072.815,A -85,B 0,C 180,E1 15043.546,E2 15043.546} C_VEL
LIN {X 0,Y 305.284,Z 1058.957,A -85,B 0,C 180,E1 15051.072,E2 15051.072} C_VEL
LIN {X 0,Y 309.568,Z 1039.672,A -85,B 0,C 180,E1 15058.313,E2 15058.313} C_VEL
LIN {X 0,Y 316.563,Z 1015.353,A -85,B 0,C 180,E1 15065.023,E2 15065.023} C_VEL
LIN {X 0,Y 326.167,Z 985.467,A -85,B 0,C 180,E1 15071.151,E2 15071.151} C_VEL
LIN {X 0,Y 329.762,Z 974.843,A -85,B 0,C 180,E1 15072.921,E2 15072.921} C_VEL
LIN {X 0,Y 330.488,Z 962.817,A -85,B 0,C 180,E1 15075.126,E2 15075.126} C_VEL
LIN {X 0,Y 331.332,Z 950.326,A -85,B 0,C 180,E1 15077.249,E2 15077.249} C_VEL
LIN {X 0,Y 343.013,Z 913.29,A -85,B 0,C 180,E1 15081.323,E2 15081.323} C_VEL
LIN {X 0,Y 353.809,Z 873.171,A -85,B 0,C 180,E1 15084.393,E2 15084.393} C_VEL
LIN {X 0,Y 358.085,Z 852.306,A -85,B 0,C 180,E1 15085.642,E2 15085.642} C_VEL
LIN {X 0,Y 349.189,Z 826.099,A -85,B 0,C 180,E1 15089.638,E2 15089.638} C_VEL
LIN {X 0,Y 336.341,Z 800.147,A -85,B 0,C 180,E1 15094.781,E2 15094.781} C_VEL
LIN {X 0,Y 323.749,Z 779.322,A -85,B 0,C 180,E1 15100.302,E2 15100.302} C_VEL
LIN {X 0,Y 314.279,Z 765.999,A -85,B 0,C 180,E1 15105.344,E2 15105.344} C_VEL
LIN {X 0,Y 309.504,Z 759.334,A -85,B 0,C 180,E1 15108.554,E2 15108.554} C_VEL
LIN {X 0,Y 305.745,Z 753.614,A -85,B 0,C 180,E1 15111.719,E2 15111.719} C_VEL
LIN {X 0,Y 300.718,Z 746.944,A -85,B 0,C 180,E1 15118.009,E2 15118.009} C_VEL
LIN {X 0,Y 300.196,Z 745.184,A -85,B 0,C 180,E1 15119.27,E2 15119.27} C_VEL
LIN {X 0,Y 299.915,Z 746.007,A -85,B 0,C 180,E1 15130.104,E2 15130.104} C_VEL
LIN {X 0,Y 302.927,Z 751.708,A -85,B 0,C 180,E1 15135.255,E2 15135.255} C_VEL
LIN {X 0,Y 305.515,Z 753.768,A -85,B 0,C 180,E1 15137.847,E2 15137.847} C_VEL
LIN {X 0,Y 309.384,Z 759.594,A -85,B 0,C 180,E1 15141.147,E2 15141.147} C_VEL
LIN {X 0,Y 311.788,Z 763.336,A -85,B 0,C 180,E1 15142.916,E2 15142.916} C_VEL
LIN {X 0,Y 316.2,Z 769.286,A -85,B 0,C 180,E1 15145.706,E2 15145.706} C_VEL
LIN {X 0,Y 324.415,Z 782.275,A -85,B 0,C 180,E1 15150.391,E2 15150.391} C_VEL
LIN {X 0,Y 334.433,Z 800.866,A -85,B 0,C 180,E1 15155.615,E2 15155.615} C_VEL
LIN {X 0,Y 343.382,Z 822.721,A -85,B 0,C 180,E1 15160.595,E2 15160.595} C_VEL
LIN {X 0,Y 350.072,Z 849.044,A -85,B 0,C 180,E1 15165.745,E2 15165.745} C_VEL
LIN {X 0,Y 349.969,Z 853.66,A -85,B 0,C 180,E1 15166.443,E2 15166.443} C_VEL
LIN {X 0,Y 339.498,Z 884.191,A -85,B 0,C 180,E1 15169.921,E2 15169.921} C_VEL
LIN {X 0,Y 328.318,Z 911.576,A -85,B 0,C 180,E1 15174.396,E2 15174.396} C_VEL
LIN {X 0,Y 317.235,Z 935.267,A -85,B 0,C 180,E1 15179.927,E2 15179.927} C_VEL
LIN {X 0,Y 308.028,Z 953.83,A -85,B 0,C 180,E1 15186.291,E2 15186.291} C_VEL
LIN {X 0,Y 301.625,Z 967.02,A -85,B 0,C 180,E1 15193.225,E2 15193.225} C_VEL
LIN {X 0,Y 297.882,Z 975.642,A -85,B 0,C 180,E1 15201.23,E2 15201.23} C_VEL
LIN {X 0,Y 297.032,Z 978.375,A -85,B 0,C 180,E1 15207.079,E2 15207.079} C_VEL
LIN {X 0,Y 297.038,Z 978.342,A -85,B 0,C 180,E1 15212.922,E2 15212.922} C_VEL
LIN {X 0,Y 298.407,Z 974.423,A -85,B 0,C 180,E1 15220.229,E2 15220.229} C_VEL
LIN {X 0,Y 302.193,Z 965.703,A -85,B 0,C 180,E1 15227.494,E2 15227.494} C_VEL
LIN {X 0,Y 308.794,Z 952.165,A -85,B 0,C 180,E1 15234.269,E2 15234.269} C_VEL
LIN {X 0,Y 317.915,Z 933.712,A -85,B 0,C 180,E1 15240.397,E2 15240.397} C_VEL
LIN {X 0,Y 328.4,Z 911.134,A -85,B 0,C 180,E1 15245.594,E2 15245.594} C_VEL
LIN {X 0,Y 339.285,Z 884.66,A -85,B 0,C 180,E1 15249.901,E2 15249.901} C_VEL
LIN {X 0,Y 349.961,Z 853.487,A -85,B 0,C 180,E1 15253.466,E2 15253.466} C_VEL
LIN {X 0,Y 349.881,Z 848.398,A -85,B 0,C 180,E1 15254.269,E2 15254.269} C_VEL
LIN {X 0,Y 343.02,Z 822.248,A -85,B 0,C 180,E1 15259.428,E2 15259.428} C_VEL
LIN {X 0,Y 334.061,Z 800.127,A -85,B 0,C 180,E1 15264.44,E2 15264.44} C_VEL
LIN {X 0,Y 323.041,Z 779.581,A -85,B 0,C 180,E1 15270.242,E2 15270.242} C_VEL
LIN {X 0,Y 313.906,Z 766.052,A -85,B 0,C 180,E1 15275.523,E2 15275.523} C_VEL
LIN {X 0,Y 309.342,Z 759.534,A -85,B 0,C 180,E1 15278.662,E2 15278.662} C_VEL
LIN {X 0,Y 305.607,Z 754.093,A -85,B 0,C 180,E1 15281.786,E2 15281.786} C_VEL
LIN {X 0,Y 303.912,Z 752.259,A -85,B 0,C 180,E1 15283.412,E2 15283.412} C_VEL
LIN {X 0,Y 300.064,Z 746.684,A -85,B 0,C 180,E1 15288.82,E2 15288.82} C_VEL
LIN {X 0,Y 299.477,Z 745.174,A -85,B 0,C 180,E1 15290.335,E2 15290.335} C_VEL
LIN {X 0,Y 300.469,Z 745.641,A -85,B 0,C 180,E1 15301.722,E2 15301.722} C_VEL
LIN {X 0,Y 302.863,Z 751.122,A -85,B 0,C 180,E1 15305.565,E2 15305.565} C_VEL
LIN {X 0,Y 305.86,Z 753.911,A -85,B 0,C 180,E1 15308.547,E2 15308.547} C_VEL
LIN {X 0,Y 310.209,Z 759.85,A -85,B 0,C 180,E1 15312.045,E2 15312.045} C_VEL
LIN {X 0,Y 317.231,Z 770.276,A -85,B 0,C 180,E1 15316.467,E2 15316.467} C_VEL
LIN {X 0,Y 325.517,Z 782.449,A -85,B 0,C 180,E1 15320.625,E2 15320.625} C_VEL
LIN {X 0,Y 337.574,Z 802.3,A -85,B 0,C 180,E1 15325.757,E2 15325.757} C_VEL
LIN {X 0,Y 350.313,Z 829.107,A -85,B 0,C 180,E1 15330.883,E2 15330.883} C_VEL
LIN {X 0,Y 358.209,Z 853.075,A -85,B 0,C 180,E1 15334.467,E2 15334.467} C_VEL
LIN {X 0,Y 348.034,Z 895.73,A -85,B 0,C 180,E1 15337.194,E2 15337.194} C_VEL
LIN {X 0,Y 336.15,Z 935.31,A -85,B 0,C 180,E1 15340.928,E2 15340.928} C_VEL
LIN {X 0,Y 324.048,Z 971.519,A -85,B 0,C 180,E1 15345.79,E2 15345.79} C_VEL
LIN {X 0,Y 313.159,Z 1003.27,A -85,B 0,C 180,E1 15351.678,E2 15351.678} C_VEL
LIN {X 0,Y 304.617,Z 1029.807,A -85,B 0,C 180,E1 15358.352,E2 15358.352} C_VEL
LIN {X 0,Y 298.931,Z 1051.393,A -85,B 0,C 180,E1 15365.741,E2 15365.741} C_VEL
LIN {X 0,Y 296.13,Z 1067.668,A -85,B 0,C 180,E1 15373.668,E2 15373.668} C_VEL
LIN {X 0,Y 295.439,Z 1075.748,A -85,B 0,C 180,E1 15379.667,E2 15379.667} C_VEL
LIN {X 0,Y 295.454,Z 1079.512,A -85,B 0,C 180,E1 15384.117,E2 15384.117} C_VEL
LIN {X 0,Y 295.698,Z 1081.381,A -85,B 0,C 180,E1 15390,E2 15390} C_VEL
LIN {X 0,Y 295.425,Z 1079.511,A -85,B 0,C 180,E1 15395.883,E2 15395.883} C_VEL
LIN {X 0,Y 295.7,Z 1072.094,A -85,B 0,C 180,E1 15403.38,E2 15403.38} C_VEL
LIN {X 0,Y 297.312,Z 1059.09,A -85,B 0,C 180,E1 15410.883,E2 15410.883} C_VEL
LIN {X 0,Y 301.717,Z 1040.065,A -85,B 0,C 180,E1 15418.428,E2 15418.428} C_VEL
LIN {X 0,Y 309.172,Z 1015.276,A -85,B 0,C 180,E1 15425.556,E2 15425.556} C_VEL
LIN {X 0,Y 318.881,Z 986.566,A -85,B 0,C 180,E1 15431.659,E2 15431.659} C_VEL
LIN {X 0,Y 330.229,Z 953.628,A -85,B 0,C 180,E1 15436.819,E2 15436.819} C_VEL
LIN {X 0,Y 331.332,Z 950.326,A -85,B 0,C 180,E1 15437.249,E2 15437.249} C_VEL
LIN {X 0,Y 332.459,Z 937.374,A -85,B 0,C 180,E1 15439.292,E2 15439.292} C_VEL
LIN {X 0,Y 333.383,Z 925.76,A -85,B 0,C 180,E1 15441.008,E2 15441.008} C_VEL
LIN {X 0,Y 333.919,Z 923.95,A -85,B 0,C 180,E1 15441.204,E2 15441.204} C_VEL
LIN {X 0,Y 345.266,Z 885.945,A -85,B 0,C 180,E1 15444.485,E2 15444.485} C_VEL
LIN {X 0,Y 352.484,Z 855.415,A -85,B 0,C 180,E1 15446.421,E2 15446.421} C_VEL
LIN {X 0,Y 343.672,Z 829.239,A -85,B 0,C 180,E1 15450.648,E2 15450.648} C_VEL
LIN {X 0,Y 331.516,Z 803.722,A -85,B 0,C 180,E1 15455.975,E2 15455.975} C_VEL
LIN {X 0,Y 320.149,Z 784.809,A -85,B 0,C 180,E1 15461.365,E2 15461.365} C_VEL
LIN {X 0,Y 312.147,Z 773.038,A -85,B 0,C 180,E1 15465.959,E2 15465.959} C_VEL
LIN {X 0,Y 307.92,Z 766.848,A -85,B 0,C 180,E1 15468.931,E2 15468.931} C_VEL
LIN {X 0,Y 303.578,Z 760.22,A -85,B 0,C 180,E1 15472.831,E2 15472.831} C_VEL
LIN {X 0,Y 299.62,Z 754.814,A -85,B 0,C 180,E1 15478.183,E2 15478.183} C_VEL
LIN {X 0,Y 298.871,Z 752.904,A -85,B 0,C 180,E1 15479.992,E2 15479.992} C_VEL
LIN {X 0,Y 298.843,Z 753.894,A -85,B 0,C 180,E1 15489.884,E2 15489.884} C_VEL
LIN {X 0,Y 302.01,Z 759.605,A -85,B 0,C 180,E1 15495.302,E2 15495.302} C_VEL
LIN {X 0,Y 304.214,Z 761.876,A -85,B 0,C 180,E1 15497.645,E2 15497.645} C_VEL
LIN {X 0,Y 309.514,Z 769.866,A -85,B 0,C 180,E1 15502.171,E2 15502.171} C_VEL
LIN {X 0,Y 315,Z 778.4,A -85,B 0,C 180,E1 15506.003,E2 15506.003} C_VEL
LIN {X 0,Y 324.087,Z 793.824,A -85,B 0,C 180,E1 15511.453,E2 15511.453} C_VEL
LIN {X 0,Y 333.598,Z 814.403,A -85,B 0,C 180,E1 15516.953,E2 15516.953} C_VEL
LIN {X 0,Y 340.731,Z 836.325,A -85,B 0,C 180,E1 15521.785,E2 15521.785} C_VEL
LIN {X 0,Y 344.506,Z 855.155,A -85,B 0,C 180,E1 15525.539,E2 15525.539} C_VEL
LIN {X 0,Y 333.561,Z 885.904,A -85,B 0,C 180,E1 15529.089,E2 15529.089} C_VEL
LIN {X 0,Y 322.035,Z 913.04,A -85,B 0,C 180,E1 15533.591,E2 15533.591} C_VEL
LIN {X 0,Y 310.848,Z 935.958,A -85,B 0,C 180,E1 15538.999,E2 15538.999} C_VEL
LIN {X 0,Y 300.902,Z 955.209,A -85,B 0,C 180,E1 15545.692,E2 15545.692} C_VEL
LIN {X 0,Y 294.141,Z 968.381,A -85,B 0,C 180,E1 15552.785,E2 15552.785} C_VEL
LIN {X 0,Y 290.185,Z 976.992,A -85,B 0,C 180,E1 15560.995,E2 15560.995} C_VEL
LIN {X 0,Y 289.27,Z 979.722,A -85,B 0,C 180,E1 15567,E2 15567} C_VEL
LIN {X 0,Y 289.277,Z 979.689,A -85,B 0,C 180,E1 15573,E2 15573} C_VEL
LIN {X 0,Y 290.728,Z 975.78,A -85,B 0,C 180,E1 15580.502,E2 15580.502} C_VEL
LIN {X 0,Y 294.741,Z 967.07,A -85,B 0,C 180,E1 15587.951,E2 15587.951} C_VEL
LIN {X 0,Y 301.708,Z 953.498,A -85,B 0,C 180,E1 15594.903,E2 15594.903} C_VEL
LIN {X 0,Y 311.683,Z 934.212,A -85,B 0,C 180,E1 15601.379,E2 15601.379} C_VEL
LIN {X 0,Y 322.867,Z 910.972,A -85,B 0,C 180,E1 15606.718,E2 15606.718} C_VEL
LIN {X 0,Y 334.815,Z 882.562,A -85,B 0,C 180,E1 15611.268,E2 15611.268} C_VEL
LIN {X 0,Y 344.479,Z 854.587,A -85,B 0,C 180,E1 15614.439,E2 15614.439} C_VEL
LIN {X 0,Y 338.914,Z 830.163,A -85,B 0,C 180,E1 15619.413,E2 15619.413} C_VEL
LIN {X 0,Y 330.782,Z 807.675,A -85,B 0,C 180,E1 15624.563,E2 15624.563} C_VEL
LIN {X 0,Y 320.243,Z 786.639,A -85,B 0,C 180,E1 15630.638,E2 15630.638} C_VEL
LIN {X 0,Y 311.425,Z 772.942,A -85,B 0,C 180,E1 15636.175,E2 15636.175} C_VEL
LIN {X 0,Y 307.403,Z 766.887,A -85,B 0,C 180,E1 15639.216,E2 15639.216} C_VEL
LIN {X 0,Y 303.849,Z 760.766,A -85,B 0,C 180,E1 15642.52,E2 15642.52} C_VEL
LIN {X 0,Y 299.011,Z 754.687,A -85,B 0,C 180,E1 15648.975,E2 15648.975} C_VEL
LIN {X 0,Y 298.545,Z 753.024,A -85,B 0,C 180,E1 15650.305,E2 15650.305} C_VEL
LIN {X 0,Y 299.313,Z 753.551,A -85,B 0,C 180,E1 15661.457,E2 15661.457} C_VEL
LIN {X 0,Y 302.009,Z 759.207,A -85,B 0,C 180,E1 15665.761,E2 15665.761} C_VEL
LIN {X 0,Y 304.436,Z 761.712,A -85,B 0,C 180,E1 15668.227,E2 15668.227} C_VEL
LIN {X 0,Y 309.853,Z 769.811,A -85,B 0,C 180,E1 15672.63,E2 15672.63} C_VEL
LIN {X 0,Y 315.364,Z 777.777,A -85,B 0,C 180,E1 15676.119,E2 15676.119} C_VEL
LIN {X 0,Y 325.758,Z 793.792,A -85,B 0,C 180,E1 15681.46,E2 15681.46} C_VEL
LIN {X 0,Y 337.615,Z 815.85,A -85,B 0,C 180,E1 15686.767,E2 15686.767} C_VEL
LIN {X 0,Y 347.62,Z 839.523,A -85,B 0,C 180,E1 15691.149,E2 15691.149} C_VEL
LIN {X 0,Y 352.408,Z 855.405,A -85,B 0,C 180,E1 15693.587,E2 15693.587} C_VEL
LIN {X 0,Y 342.024,Z 897.327,A -85,B 0,C 180,E1 15696.382,E2 15696.382} C_VEL
LIN {X 0,Y 330.005,Z 935.551,A -85,B 0,C 180,E1 15700.065,E2 15700.065} C_VEL
LIN {X 0,Y 317.971,Z 969.919,A -85,B 0,C 180,E1 15704.734,E2 15704.734} C_VEL
LIN {X 0,Y 306.819,Z 1001.037,A -85,B 0,C 180,E1 15710.557,E2 15710.557} C_VEL
LIN {X 0,Y 297.386,Z 1028.572,A -85,B 0,C 180,E1 15717.593,E2 15717.593} C_VEL
LIN {X 0,Y 291.179,Z 1050.725,A -85,B 0,C 180,E1 15725.42,E2 15725.42} C_VEL
LIN {X 0,Y 288.358,Z 1066.244,A -85,B 0,C 180,E1 15733.215,E2 15733.215} C_VEL
LIN {X 0,Y 287.621,Z 1074.363,A -85,B 0,C 180,E1 15739.383,E2 15739.383} C_VEL
LIN {X 0,Y 287.643,Z 1078.148,A -85,B 0,C 180,E1 15743.957,E2 15743.957} C_VEL
LIN {X 0,Y 287.922,Z 1080.034,A -85,B 0,C 180,E1 15750,E2 15750} C_VEL
LIN {X 0,Y 287.621,Z 1078.148,A -85,B 0,C 180,E1 15756.043,E2 15756.043} C_VEL
LIN {X 0,Y 287.918,Z 1070.696,A -85,B 0,C 180,E1 15763.748,E2 15763.748} C_VEL
LIN {X 0,Y 289.651,Z 1057.634,A -85,B 0,C 180,E1 15771.462,E2 15771.462} C_VEL
LIN {X 0,Y 294.355,Z 1038.452,A -85,B 0,C 180,E1 15779.24,E2 15779.24} C_VEL
LIN {X 0,Y 302.272,Z 1013.691,A -85,B 0,C 180,E1 15786.497,E2 15786.497} C_VEL
LIN {X 0,Y 312.637,Z 984.934,A -85,B 0,C 180,E1 15792.685,E2 15792.685} C_VEL
LIN {X 0,Y 324.734,Z 951.289,A -85,B 0,C 180,E1 15797.982,E2 15797.982} C_VEL
LIN {X 0,Y 333.919,Z 923.95,A -85,B 0,C 180,E1 15801.204,E2 15801.204} C_VEL
LIN {X 0,Y 335.513,Z 910.066,A -85,B 0,C 180,E1 15803.021,E2 15803.021} C_VEL
LIN {X 0,Y 337.133,Z 895.779,A -85,B 0,C 180,E1 15804.723,E2 15804.723} C_VEL
LIN {X 0,Y 346.852,Z 858.42,A -85,B 0,C 180,E1 15807.235,E2 15807.235} C_VEL
LIN {X 0,Y 338.113,Z 831.949,A -85,B 0,C 180,E1 15811.768,E2 15811.768} C_VEL
LIN {X 0,Y 327.037,Z 808.133,A -85,B 0,C 180,E1 15817.033,E2 15817.033} C_VEL
LIN {X 0,Y 315.474,Z 787.748,A -85,B 0,C 180,E1 15823.167,E2 15823.167} C_VEL
LIN {X 0,Y 306.172,Z 774.27,A -85,B 0,C 180,E1 15829.397,E2 15829.397} C_VEL
LIN {X 0,Y 301.877,Z 767.703,A -85,B 0,C 180,E1 15833.514,E2 15833.514} C_VEL
LIN {X 0,Y 298.308,Z 761.849,A -85,B 0,C 180,E1 15838.902,E2 15838.902} C_VEL
LIN {X 0,Y 297.374,Z 760.659,A -85,B 0,C 180,E1 15841.451,E2 15841.451} C_VEL
LIN {X 0,Y 297.77,Z 761.644,A -85,B 0,C 180,E1 15849.615,E2 15849.615} C_VEL
LIN {X 0,Y 300.927,Z 767.485,A -85,B 0,C 180,E1 15855.359,E2 15855.359} C_VEL
LIN {X 0,Y 302.655,Z 769.364,A -85,B 0,C 180,E1 15857.249,E2 15857.249} C_VEL
LIN {X 0,Y 307.709,Z 777.828,A -85,B 0,C 180,E1 15862.025,E2 15862.025} C_VEL
LIN {X 0,Y 312.415,Z 785.473,A -85,B 0,C 180,E1 15865.559,E2 15865.559} C_VEL
LIN {X 0,Y 321.017,Z 801.029,A -85,B 0,C 180,E1 15871.151,E2 15871.151} C_VEL
LIN {X 0,Y 330.287,Z 822.931,A -85,B 0,C 180,E1 15877.099,E2 15877.099} C_VEL
LIN {X 0,Y 336.403,Z 845.451,A -85,B 0,C 180,E1 15882.109,E2 15882.109} C_VEL
LIN {X 0,Y 338.553,Z 858.331,A -85,B 0,C 180,E1 15884.767,E2 15884.767} C_VEL
LIN {X 0,Y 327.263,Z 888.664,A -85,B 0,C 180,E1 15888.374,E2 15888.374} C_VEL
LIN {X 0,Y 314.896,Z 916.512,A -85,B 0,C 180,E1 15893.162,E2 15893.162} C_VEL
LIN {X 0,Y 302.576,Z 940.492,A -85,B 0,C 180,E1 15899.174,E2 15899.174} C_VEL
LIN {X 0,Y 293.148,Z 957.737,A -85,B 0,C 180,E1 15905.596,E2 15905.596} C_VEL
LIN {X 0,Y 286.147,Z 970.733,A -85,B 0,C 180,E1 15913.082,E2 15913.082} C_VEL
LIN {X 0,Y 282.485,Z 978.344,A -85,B 0,C 180,E1 15920.748,E2 15920.748} C_VEL
LIN {X 0,Y 281.501,Z 981.069,A -85,B 0,C 180,E1 15926.917,E2 15926.917} C_VEL
LIN {X 0,Y 281.508,Z 981.036,A -85,B 0,C 180,E1 15933.083,E2 15933.083} C_VEL
LIN {X 0,Y 283.06,Z 977.136,A -85,B 0,C 180,E1 15940.79,E2 15940.79} C_VEL
LIN {X 0,Y 287.444,Z 968.199,A -85,B 0,C 180,E1 15948.584,E2 15948.584} C_VEL
LIN {X 0,Y 294.878,Z 954.407,A -85,B 0,C 180,E1 15955.743,E2 15955.743} C_VEL
LIN {X 0,Y 304.798,Z 936.108,A -85,B 0,C 180,E1 15962.004,E2 15962.004} C_VEL
LIN {X 0,Y 316.516,Z 912.756,A -85,B 0,C 180,E1 15967.497,E2 15967.497} C_VEL
LIN {X 0,Y 329.057,Z 884.082,A -85,B 0,C 180,E1 15972.162,E2 15972.162} C_VEL
LIN {X 0,Y 338.41,Z 857.153,A -85,B 0,C 180,E1 15975.344,E2 15975.344} C_VEL
LIN {X 0,Y 333.169,Z 832.531,A -85,B 0,C 180,E1 15980.581,E2 15980.581} C_VEL
LIN {X 0,Y 325.714,Z 811.506,A -85,B 0,C 180,E1 15985.707,E2 15985.707} C_VEL
LIN {X 0,Y 316.453,Z 792.4,A -85,B 0,C 180,E1 15991.581,E2 15991.581} C_VEL
LIN {X 0,Y 309.023,Z 779.935,A -85,B 0,C 180,E1 15996.744,E2 15996.744} C_VEL
LIN {X 0,Y 305.407,Z 774.219,A -85,B 0,C 180,E1 15999.705,E2 15999.705} C_VEL
LIN {X 0,Y 301.512,Z 767.803,A -85,B 0,C 180,E1 16003.696,E2 16003.696} C_VEL
LIN {X 0,Y 297.822,Z 761.838,A -85,B 0,C 180,E1 16009.593,E2 16009.593} C_VEL
LIN {X 0,Y 296.645,Z 760.497,A -85,B 0,C 180,E1 16014.15,E2 16014.15} C_VEL
LIN {X 0,Y 298.207,Z 761.53,A -85,B 0,C 180,E1 16021.28,E2 16021.28} C_VEL
LIN {X 0,Y 301.17,Z 767.206,A -85,B 0,C 180,E1 16025.958,E2 16025.958} C_VEL
LIN {X 0,Y 303.031,Z 769.441,A -85,B 0,C 180,E1 16027.904,E2 16027.904} C_VEL
LIN {X 0,Y 308.2,Z 777.459,A -85,B 0,C 180,E1 16032.327,E2 16032.327} C_VEL
LIN {X 0,Y 315.736,Z 788.462,A -85,B 0,C 180,E1 16037.093,E2 16037.093} C_VEL
LIN {X 0,Y 327.873,Z 809.657,A -85,B 0,C 180,E1 16043.423,E2 16043.423} C_VEL
LIN {X 0,Y 339.685,Z 835.86,A -85,B 0,C 180,E1 16048.998,E2 16048.998} C_VEL
LIN {X 0,Y 346.703,Z 858.109,A -85,B 0,C 180,E1 16052.729,E2 16052.729} C_VEL
LIN {X 0,Y 336.589,Z 897.126,A -85,B 0,C 180,E1 16055.386,E2 16055.386} C_VEL
LIN {X 0,Y 324.68,Z 933.777,A -85,B 0,C 180,E1 16058.934,E2 16058.934} C_VEL
LIN {X 0,Y 311.629,Z 969.339,A -85,B 0,C 180,E1 16063.806,E2 16063.806} C_VEL
LIN {X 0,Y 299.713,Z 1001.09,A -85,B 0,C 180,E1 16069.904,E2 16069.904} C_VEL
LIN {X 0,Y 290.026,Z 1027.901,A -85,B 0,C 180,E1 16076.972,E2 16076.972} C_VEL
LIN {X 0,Y 283.662,Z 1049.25,A -85,B 0,C 180,E1 16084.723,E2 16084.723} C_VEL
LIN {X 0,Y 280.615,Z 1064.825,A -85,B 0,C 180,E1 16092.738,E2 16092.738} C_VEL
LIN {X 0,Y 279.806,Z 1072.977,A -85,B 0,C 180,E1 16099.083,E2 16099.083} C_VEL
LIN {X 0,Y 279.843,Z 1076.785,A -85,B 0,C 180,E1 16103.788,E2 16103.788} C_VEL
LIN {X 0,Y 280.157,Z 1078.689,A -85,B 0,C 180,E1 16110,E2 16110} C_VEL
LIN {X 0,Y 279.822,Z 1076.786,A -85,B 0,C 180,E1 16116.212,E2 16116.212} C_VEL
LIN {X 0,Y 280.017,Z 1070.345,A -85,B 0,C 180,E1 16123.274,E2 16123.274} C_VEL
LIN {X 0,Y 281.585,Z 1058.252,A -85,B 0,C 180,E1 16131.031,E2 16131.031} C_VEL
LIN {X 0,Y 286.272,Z 1039.634,A -85,B 0,C 180,E1 16139.112,E2 16139.112} C_VEL
LIN {X 0,Y 294.793,Z 1014.071,A -85,B 0,C 180,E1 16146.98,E2 16146.98} C_VEL
LIN {X 0,Y 305.764,Z 985.184,A -85,B 0,C 180,E1 16153.409,E2 16153.409} C_VEL
LIN {X 0,Y 318.517,Z 951.335,A -85,B 0,C 180,E1 16158.869,E2 16158.869} C_VEL
